// TIA Portal V18 program export: 1 tag tables, 1 data types, 4 data blocks, 17 code blocks (in call order from the OBs), 10 instance data blocks

VAR_GLOBAL   // PLC tag table "默认变量表"
   System_Byte AT %MB1 : Byte;
   FirstScan AT %M1.0 : Bool;
   DiagStatusUpdate AT %M1.1 : Bool;
   AlwaysTRUE AT %M1.2 : Bool;
   AlwaysFALSE AT %M1.3 : Bool;
   Clock_Byte AT %MB0 : Byte;
   Clock_10Hz AT %M0.0 : Bool;
   Clock_5Hz AT %M0.1 : Bool;
   "Clock_2.5Hz" AT %M0.2 : Bool;
   Clock_2Hz AT %M0.3 : Bool;
   "Clock_1.25Hz" AT %M0.4 : Bool;
   Clock_1Hz AT %M0.5 : Bool;
   "Clock_0.625Hz" AT %M0.6 : Bool;
   "Clock_0.5Hz" AT %M0.7 : Bool;
END_VAR

TYPE "FIODia"
// stored: IsFailsafeCompliant true
   STRUCT
      ModulePassOut : Bool;   // 模块钝化
      ModuleACK_REQ : Bool;   // 模块需确认重新集成
      Channel0PassOut : Bool;   // 通道0钝化
      Channel1PassOut : Bool;   // 通道1钝化
      Channel2PassOut : Bool;   // 通道2钝化
      Channel3PassOut : Bool;   // 通道3钝化
      Channel4PassOut : Bool;   // 通道4钝化
      Channel5PassOut : Bool;   // 通道5钝化
      Channel6PassOut : Bool;   // 通道6钝化
      Channel7PassOut : Bool;   // 通道7钝化
   END_STRUCT;
END_TYPE

DATA_BLOCK "TCSData"   // DB4
{ S7_Optimized_Access := 'TRUE' }
VERSION : 0.1
// stored: AutoNumber true, DBAccessibleFromOPCUA true, IsOnlyStoredInLoadMemory false, IsRetainMemResEnabled false, IsWriteProtectedInAS false, MemoryReserve 100
   VAR
      Data : Array[0..1] of Word;
      Connect : TCON_IP_v4;
   END_VAR
BEGIN
   Connect.InterfaceId := 64;
   Connect.ID := 16#1;
   Connect.LocalPort := 502;
END_DATA_BLOCK

DATA_BLOCK "数据块_1"   // DB2
{ S7_Optimized_Access := 'TRUE' }
VERSION : 0.1
// stored: AutoNumber true, DBAccessibleFromOPCUA true, IsOnlyStoredInLoadMemory false, IsRetainMemResEnabled false, IsWriteProtectedInAS false, MemoryReserve 100
   VAR
      Room1_Interlock : Bool;
      Room2_Interlock : Bool;
      ACC_Interlock : Bool;
      VerticalBeam_Interlock : Bool;
      Interlock : Bool;
   END_VAR
BEGIN
END_DATA_BLOCK

DATA_BLOCK "数据块_2"   // DB3
{ S7_Optimized_Access := 'TRUE' }
VERSION : 0.1
// stored: AutoNumber true, DBAccessibleFromOPCUA true, IsOnlyStoredInLoadMemory false, IsRetainMemResEnabled false, IsWriteProtectedInAS false, MemoryReserve 100
   VAR
      "F-DI_A21_1" : "FIODia";   // 安全输入模块A21.1
      "F-DI_A21_2" { S7_SetPoint := 'True'} : "FIODia";   // 安全输入模块A21.2
      "F-DI_A21_3" { S7_SetPoint := 'True'} : "FIODia";   // 安全输入模块A21.3
      "F-DI_A21_4" { S7_SetPoint := 'True'} : "FIODia";   // 安全输入模块A21.4
      "F-DI_A21_5" { S7_SetPoint := 'True'} : "FIODia";   // 安全输入模块A21.5
      "F-DI_A21_6" { S7_SetPoint := 'True'} : "FIODia";   // 安全输入模块A21.6
      "F-DI_A21_7" { S7_SetPoint := 'True'} : "FIODia";   // 安全输入模块A21.7
      "F-DI_A21_8" { S7_SetPoint := 'True'} : "FIODia";   // 安全输入模块A21.8
      "F-DI_A21_9" { S7_SetPoint := 'True'} : "FIODia";   // 安全输入模块A21.9
      "F-DI_A21_10" { S7_SetPoint := 'True'} : "FIODia";   // 安全输入模块A21.10
      "F-DI_A21_11" { S7_SetPoint := 'True'} : "FIODia";   // 安全输入模块A21.11
      "F-DI_A21_12" { S7_SetPoint := 'True'} : "FIODia";   // 安全输入模块A21.12
      "F-DQ_A21_1" { S7_SetPoint := 'True'} : "FIODia";   // 安全输出模块A22.1
      "F-DQ_A21_2" { S7_SetPoint := 'True'} : "FIODia";   // 安全输出模块A22.2
   END_VAR
BEGIN
END_DATA_BLOCK

DATA_BLOCK "EPICSData"   // DB8
{ S7_Optimized_Access := 'FALSE'; DB_Accessible_From_OPC_UA := 'FALSE' }
VERSION : 0.1
// stored: AutoNumber true, DBAccessibleFromOPCUA false, IsOnlyStoredInLoadMemory false, IsWriteProtectedInAS false
   VAR
      Reset : Bool;
   END_VAR
BEGIN
END_DATA_BLOCK

ORGANIZATION_BLOCK "Main"   // OB1, LAD, ProgramCycle
TITLE = "Main Program Sweep (Cycle)"
{ S7_Optimized_Access := 'TRUE' }
VERSION : 0.1
// stored: AutoNumber true, IsIECCheckEnabled false, SetENOAutomatically false
   VAR_INPUT
      Initial_Call : Bool;   // Initial call of this OB
      Remanence : Bool;   // =True, if remanent data are available
   END_VAR
BEGIN

REGION Network 1: 11
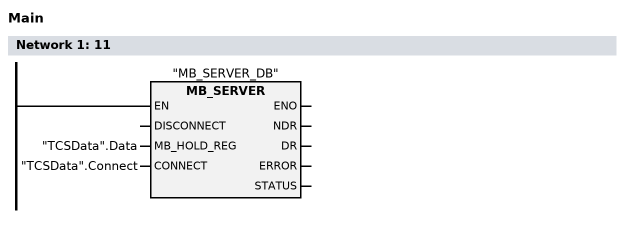
   RUNG wire#powerrail
      "MB_SERVER_DB".MB_SERVER(DISCONNECT :=, MB_HOLD_REG := "TCSData".Data, CONNECT := "TCSData".Connect, NDR =>, DR =>, ERROR =>, STATUS =>)
   END_RUNG
   // the same network as SCL:
   "MB_SERVER_DB"(MB_HOLD_REG := "TCSData".Data, CONNECT := "TCSData".Connect);   // MB_SERVER
END_REGION
END_ORGANIZATION_BLOCK

ORGANIZATION_BLOCK "Time error interrupt"   // OB80, LAD, TimeErrorInterrupt
{ S7_Optimized_Access := 'TRUE' }
VERSION : 0.1
// stored: IsIECCheckEnabled false, SetENOAutomatically false
   VAR_INPUT
      Fault_ID : Byte;   // Fault identifier
      Csg_OBnr : OB_ANY;   // Number of OB causing the error
      Csg_Prio : UInt;   // Priority of OB causing the error
   END_VAR
BEGIN
END_ORGANIZATION_BLOCK

FUNCTION_BLOCK "AccessControl"   // FB7, LAD
{ S7_Optimized_Access := 'TRUE' }
VERSION : 0.1
// stored: AutoNumber true, IsIECCheckEnabled false, IsRetainMemResEnabled false, MemoryReserve 100, SetENOAutomatically false, UDAEnableTagReadback false
   VAR_INPUT
      SearchStatus : Int;   // 0:未搜索;1:搜索中;2:搜索完成;
      RunArea : Bool;
      ACC_Ready : Bool;
      ACC_Run : Bool;
      ACC_StopBeam : Bool;
      Key : Bool;
      keyControl : Bool;
      Interlock : Bool;
      DoseAttenuation_Time : Time := T#1m;
      StartAlarm_Time : Time := T#2m;
   END_VAR
   VAR_OUTPUT
      StartAlarm : Bool;
      NoEntry : Bool;
      RestrictedEntry : Bool;
      ControlEntry : Bool;
   END_VAR
   VAR_IN_OUT
      AreaReady : Bool;
      BeamAllowed : Bool;
   END_VAR
   VAR
      State : Int;   // 0:禁止进入;1:限制进入;2:控制进入
      DoseAttenuation_Timer { S7_SetPoint := 'True'} : TON_TIME;
      StartAlarm_Timer { S7_SetPoint := 'True'} : TON_TIME;
   END_VAR
   VAR_TEMP   // added for the SCL form of the ladder/FBD networks
      _w1 : Bool;
   END_VAR
BEGIN

REGION Network 1
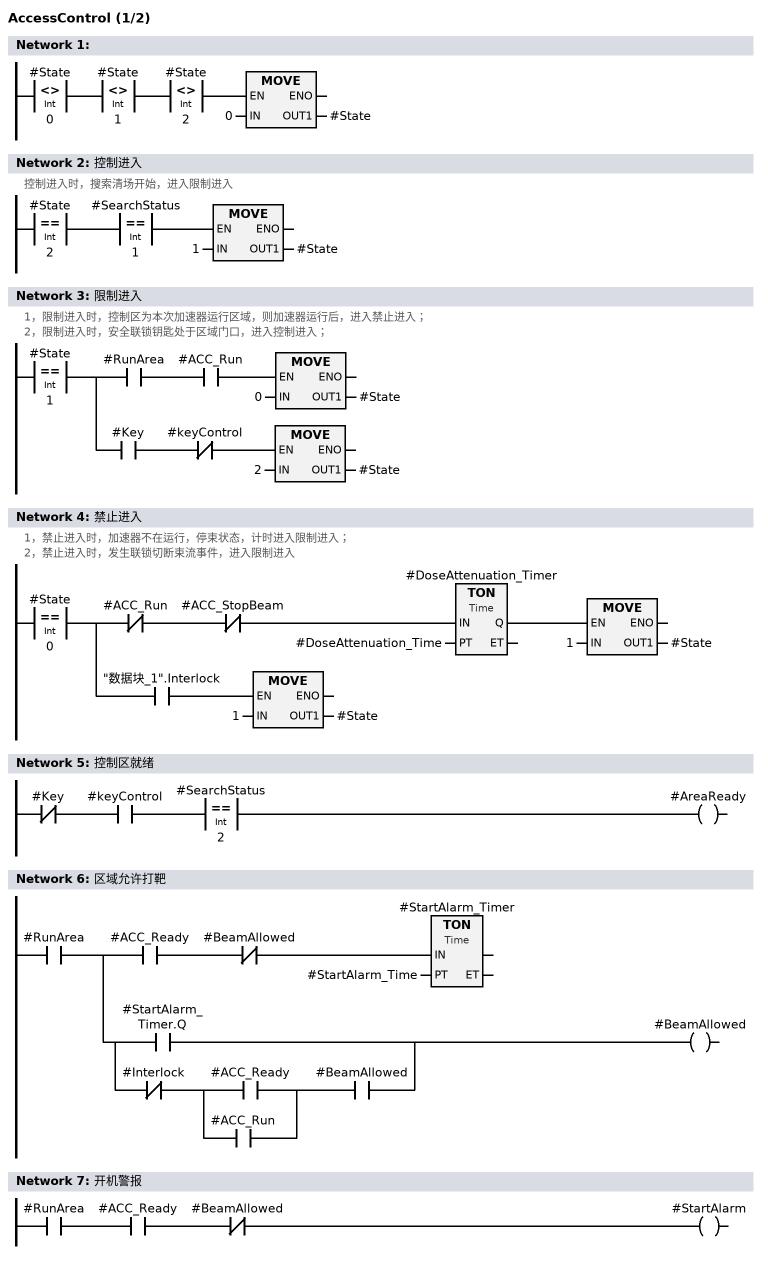
   RUNG wire#powerrail
      { S7_Templates := "SrcType := Int" } NE_Contact(in1 := #State, in2 := 0)
      { S7_Templates := "SrcType := Int" } NE_Contact(in1 := #State, in2 := 1)
      { S7_Templates := "SrcType := Int" } NE_Contact(in1 := #State, in2 := 2)
      Move(in := 0, out1 => #State)
   END_RUNG
   // the same network as SCL:
   IF (#State <> 0) AND (#State <> 1) AND (#State <> 2) THEN #State := 0; END_IF;
END_REGION

REGION Network 2: 控制进入
   // 控制进入时，搜索清场开始，进入限制进入
   RUNG wire#powerrail
      { S7_Templates := "SrcType := Int" } EQ_Contact(in1 := #State, in2 := 2)
      { S7_Templates := "SrcType := Int" } EQ_Contact(in1 := #SearchStatus, in2 := 1)
      Move(in := 1, out1 => #State)
   END_RUNG
   // the same network as SCL:
   IF (#State = 2) AND (#SearchStatus = 1) THEN #State := 1; END_IF;
END_REGION

REGION Network 3: 限制进入
   // 1，限制进入时，控制区为本次加速器运行区域，则加速器运行后，进入禁止进入；
   // 2，限制进入时，安全联锁钥匙处于区域门口，进入控制进入；
   RUNG wire#powerrail
      { S7_Templates := "SrcType := Int" } EQ_Contact(in1 := #State, in2 := 1)
      wire#w1
      Contact( #RunArea )
      Contact( #ACC_Run )
      Move(in := 0, out1 => #State)
   END_RUNG
   RUNG wire#w1
      Contact( #Key )
      I_Contact( #keyControl )
      Move(in := 2, out1 => #State)
   END_RUNG
   // the same network as SCL:
   #_w1 := #State = 1;
   IF #_w1 AND #RunArea AND #ACC_Run THEN #State := 0; END_IF;
   IF #_w1 AND #Key AND NOT #keyControl THEN #State := 2; END_IF;
END_REGION

REGION Network 4: 禁止进入
   // 1，禁止进入时，加速器不在运行，停束状态，计时进入限制进入；
   // 2，禁止进入时，发生联锁切断束流事件，进入限制进入
   RUNG wire#powerrail
      { S7_Templates := "SrcType := Int" } EQ_Contact(in1 := #State, in2 := 0)
      wire#w1
      I_Contact( #ACC_Run )
      I_Contact( #ACC_StopBeam )
      { S7_Templates := "time_type := Time" } #DoseAttenuation_Timer.TON(pt := #DoseAttenuation_Time, et =>)
      Move(in := 1, out1 => #State)
   END_RUNG
   RUNG wire#w1
      Contact( "数据块_1".Interlock )
      Move(in := 1, out1 => #State)
   END_RUNG
   // the same network as SCL:
   #_w1 := #State = 0;
   #DoseAttenuation_Timer(IN := #_w1 AND NOT #ACC_Run AND NOT #ACC_StopBeam, PT := #DoseAttenuation_Time);   // TON
   IF #DoseAttenuation_Timer.Q THEN #State := 1; END_IF;
   IF #_w1 AND "数据块_1".Interlock THEN #State := 1; END_IF;
END_REGION

REGION Network 5: 控制区就绪
   RUNG wire#powerrail
      I_Contact( #Key )
      Contact( #keyControl )
      { S7_Templates := "SrcType := Int" } EQ_Contact(in1 := #SearchStatus, in2 := 2)
      Coil( #AreaReady )
   END_RUNG
   // the same network as SCL:
   #AreaReady := NOT #Key AND #keyControl AND (#SearchStatus = 2);
END_REGION

REGION Network 6: 区域允许打靶
   RUNG wire#powerrail
      Contact( #RunArea )
      wire#w1
      Contact( #ACC_Ready )
      I_Contact( #BeamAllowed )
      { S7_Templates := "time_type := Time" } #StartAlarm_Timer.TON(pt := #StartAlarm_Time, et =>)
   END_RUNG
   RUNG wire#w1
      Contact( #StartAlarm_Timer.Q )
      wire#w2
      Coil( #BeamAllowed )
   END_RUNG
   RUNG wire#w1
      I_Contact( #Interlock )
      wire#w3
      Contact( #ACC_Ready )
      wire#w4
      Contact( #BeamAllowed )
   END_RUNG wire#w2
   RUNG wire#w3
      Contact( #ACC_Run )
   END_RUNG wire#w4
   // the same network as SCL:
   #StartAlarm_Timer(IN := #RunArea AND #ACC_Ready AND NOT #BeamAllowed, PT := #StartAlarm_Time);   // TON
   #BeamAllowed := #RunArea AND (#StartAlarm_Timer.Q OR (NOT #Interlock AND (#ACC_Ready OR #ACC_Run) AND #BeamAllowed));
END_REGION

REGION Network 7: 开机警报
   RUNG wire#powerrail
      Contact( #RunArea )
      Contact( #ACC_Ready )
      I_Contact( #BeamAllowed )
      Coil( #StartAlarm )
   END_RUNG
   // the same network as SCL:
   #StartAlarm := #RunArea AND #ACC_Ready AND NOT #BeamAllowed;
END_REGION

REGION Network 8
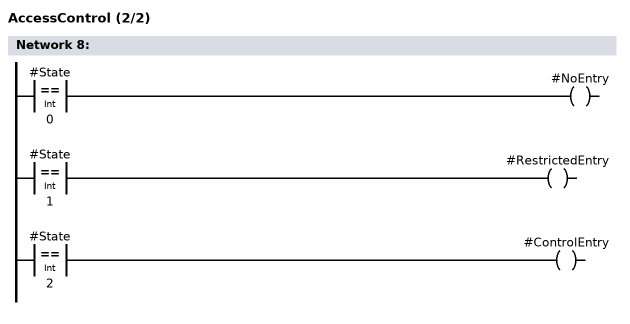
   RUNG wire#powerrail
      { S7_Templates := "SrcType := Int" } EQ_Contact(in1 := #State, in2 := 0)
      Coil( #NoEntry )
   END_RUNG
   RUNG wire#powerrail
      { S7_Templates := "SrcType := Int" } EQ_Contact(in1 := #State, in2 := 1)
      Coil( #RestrictedEntry )
   END_RUNG
   RUNG wire#powerrail
      { S7_Templates := "SrcType := Int" } EQ_Contact(in1 := #State, in2 := 2)
      Coil( #ControlEntry )
   END_RUNG
   // the same network as SCL:
   #NoEntry := #State = 0;
   #RestrictedEntry := #State = 1;
   #ControlEntry := #State = 2;
END_REGION
END_FUNCTION_BLOCK

FUNCTION_BLOCK "SearchArea"   // FB6, LAD
{ S7_Optimized_Access := 'TRUE' }
VERSION : 0.1
// stored: AutoNumber true, IsIECCheckEnabled false, IsRetainMemResEnabled false, MemoryReserve 100, SetENOAutomatically false, UDAEnableTagReadback false
   VAR_INPUT
      SB1 : Bool;
      SB2 : Bool;
      Door : Bool;
      "E-Stop" : Bool;
      SearchArea_Time : Time := T#5m;
      Reset : Bool;
   END_VAR
   VAR
      SearchArea_Timer { S7_SetPoint := 'True'} : TON_TIME;
      SearchArea_Status : Int;   // 0:未搜索;1:搜索中;2:搜索完成;
      "Step" { S7_SetPoint := 'True'} : Int;
      Error { ExternalAccessible := 'False'; ExternalVisible := 'False'; ExternalWritable := 'False'} : Struct
         All { ExternalAccessible := 'False'; ExternalVisible := 'False'; ExternalWritable := 'False'} : Bool;   // 搜索总故障
         StartFail { ExternalAccessible := 'False'; ExternalVisible := 'False'; ExternalWritable := 'False'} : Bool;   // 搜索启动失败，请确认未按下搜索按钮2或未关闭门
         WrongSequence1 { ExternalAccessible := 'False'; ExternalVisible := 'False'; ExternalWritable := 'False'} : Bool;   // 搜索顺序错误，此时应按下搜索按钮2，请勿按搜索按钮1或关闭门
         WrongSequence2 { ExternalAccessible := 'False'; ExternalVisible := 'False'; ExternalWritable := 'False'} : Bool;   // 搜索顺序错误，此时应关闭门，请勿按搜索按钮1或搜索按钮2
         Timeout { ExternalAccessible := 'False'; ExternalVisible := 'False'; ExternalWritable := 'False'} : Bool;   // 搜索超时
      END_STRUCT;
   END_VAR
   VAR_TEMP   // added for the SCL form of the ladder/FBD networks
      _w1 : Bool;
   END_VAR
BEGIN

REGION Network 1: 搜索破坏
   // 搜索完成后，当搜索按钮按下，门被打开，急停按钮按下，搜索状态设置为未搜索
   // 需与客户确认破坏条件是否包含搜索按钮和急停？
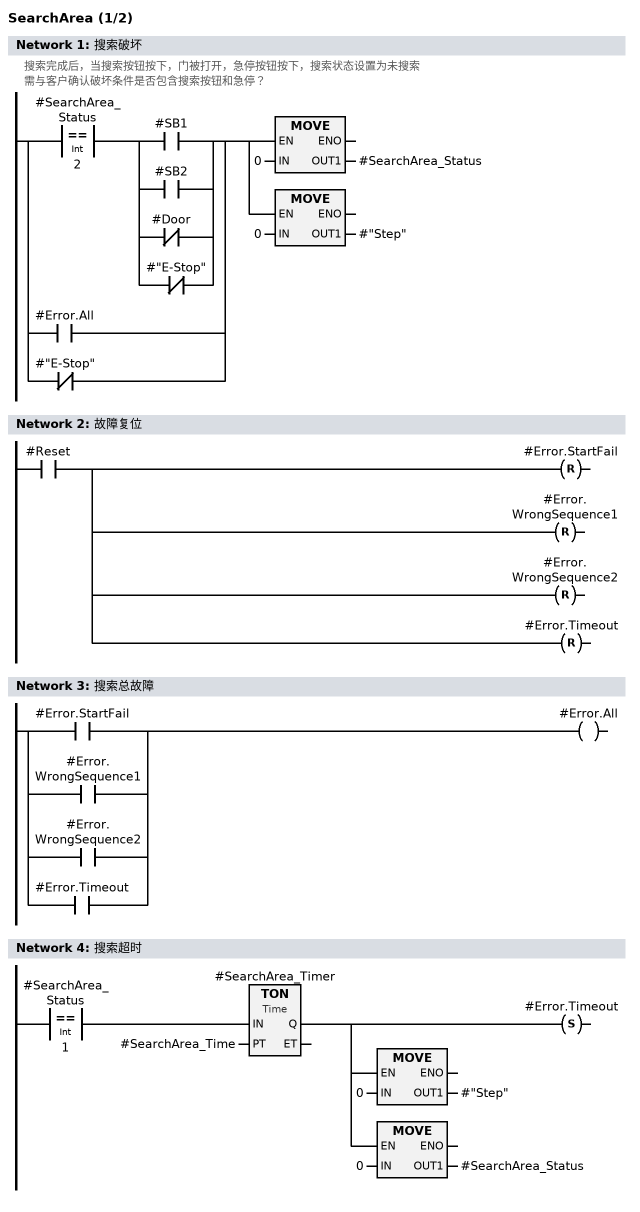
   RUNG wire#powerrail
      { S7_Templates := "SrcType := Int" } EQ_Contact(in1 := #SearchArea_Status, in2 := 2)
      wire#w1
      Contact( #SB1 )
      wire#w2
      Move(in := 0, out1 => #SearchArea_Status)
   END_RUNG
   RUNG wire#w1
      Contact( #SB2 )
   END_RUNG wire#w2
   RUNG wire#w1
      I_Contact( #Door )
   END_RUNG wire#w2
   RUNG wire#w1
      I_Contact( #"E-Stop" )
   END_RUNG wire#w2
   RUNG wire#powerrail
      Contact( #Error.All )
   END_RUNG wire#w2
   RUNG wire#powerrail
      I_Contact( #"E-Stop" )
   END_RUNG wire#w2
   RUNG wire#w2
      Move(in := 0, out1 => #"Step")
   END_RUNG
   // the same network as SCL:
   #_w1 := ((#SearchArea_Status = 2) AND (#SB1 OR #SB2 OR NOT #Door OR NOT #"E-Stop")) OR #Error.All OR NOT #"E-Stop";
   IF #_w1 THEN
       #SearchArea_Status := 0;
       #"Step" := 0;
   END_IF;
END_REGION

REGION Network 2: 故障复位
   RUNG wire#powerrail
      Contact( #Reset )
      wire#w1
      R_Coil( #Error.StartFail )
   END_RUNG
   RUNG wire#w1
      R_Coil( #Error.WrongSequence1 )
   END_RUNG
   RUNG wire#w1
      R_Coil( #Error.WrongSequence2 )
   END_RUNG
   RUNG wire#w1
      R_Coil( #Error.Timeout )
   END_RUNG
   // the same network as SCL:
   IF #Reset THEN
       #Error.StartFail := FALSE;
       #Error.WrongSequence1 := FALSE;
       #Error.WrongSequence2 := FALSE;
       #Error.Timeout := FALSE;
   END_IF;
END_REGION

REGION Network 3: 搜索总故障
   RUNG wire#powerrail
      Contact( #Error.StartFail )
      wire#w1
      Coil( #Error.All )
   END_RUNG
   RUNG wire#powerrail
      Contact( #Error.WrongSequence1 )
   END_RUNG wire#w1
   RUNG wire#powerrail
      Contact( #Error.WrongSequence2 )
   END_RUNG wire#w1
   RUNG wire#powerrail
      Contact( #Error.Timeout )
   END_RUNG wire#w1
   // the same network as SCL:
   #Error.All := #Error.StartFail OR #Error.WrongSequence1 OR #Error.WrongSequence2 OR #Error.Timeout;
END_REGION

REGION Network 4: 搜索超时
   RUNG wire#powerrail
      { S7_Templates := "SrcType := Int" } EQ_Contact(in1 := #SearchArea_Status, in2 := 1)
      { S7_Templates := "time_type := Time" } #SearchArea_Timer.TON(pt := #SearchArea_Time, et =>)
      wire#w1
      S_Coil( #Error.Timeout )
   END_RUNG
   RUNG wire#w1
      Move(in := 0, out1 => #"Step")
   END_RUNG
   RUNG wire#w1
      Move(in := 0, out1 => #SearchArea_Status)
   END_RUNG
   // the same network as SCL:
   #SearchArea_Timer(IN := #SearchArea_Status = 1, PT := #SearchArea_Time);   // TON
   IF #SearchArea_Timer.Q THEN
       #Error.Timeout := TRUE;
       #"Step" := 0;
       #SearchArea_Status := 0;
   END_IF;
END_REGION

REGION Network 5: 按下SB1，开始搜索
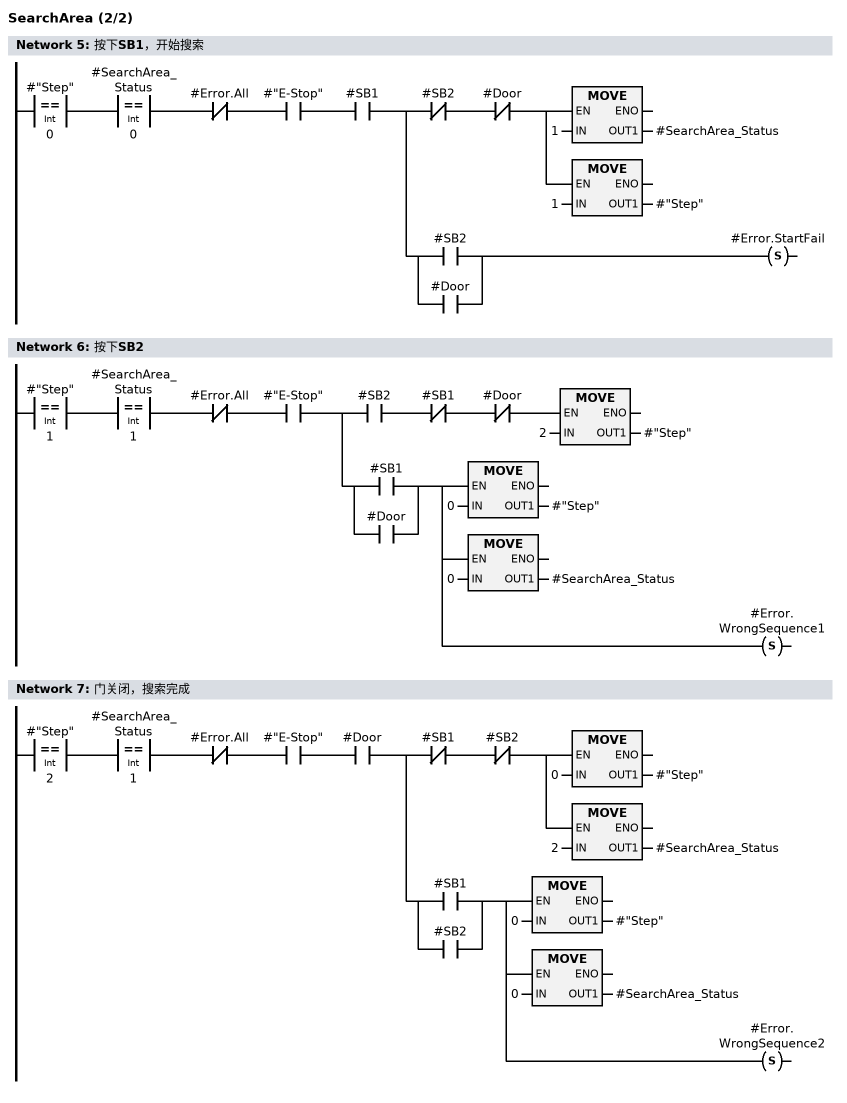
   RUNG wire#powerrail
      { S7_Templates := "SrcType := Int" } EQ_Contact(in1 := #"Step", in2 := 0)
      { S7_Templates := "SrcType := Int" } EQ_Contact(in1 := #SearchArea_Status, in2 := 0)
      I_Contact( #Error.All )
      Contact( #"E-Stop" )
      Contact( #SB1 )
      wire#w1
      I_Contact( #SB2 )
      I_Contact( #Door )
      wire#w2
      Move(in := 1, out1 => #SearchArea_Status)
   END_RUNG
   RUNG wire#w2
      Move(in := 1, out1 => #"Step")
   END_RUNG
   RUNG wire#w1
      Contact( #SB2 )
      wire#w3
      S_Coil( #Error.StartFail )
   END_RUNG
   RUNG wire#w1
      Contact( #Door )
   END_RUNG wire#w3
   // the same network as SCL:
   #_w1 := (#"Step" = 0) AND (#SearchArea_Status = 0) AND NOT #Error.All AND #"E-Stop" AND #SB1;
   IF #_w1 AND NOT #SB2 AND NOT #Door THEN
       #SearchArea_Status := 1;
       #"Step" := 1;
   END_IF;
   IF #_w1 AND (#SB2 OR #Door) THEN #Error.StartFail := TRUE; END_IF;
END_REGION

REGION Network 6: 按下SB2
   RUNG wire#powerrail
      { S7_Templates := "SrcType := Int" } EQ_Contact(in1 := #"Step", in2 := 1)
      { S7_Templates := "SrcType := Int" } EQ_Contact(in1 := #SearchArea_Status, in2 := 1)
      I_Contact( #Error.All )
      Contact( #"E-Stop" )
      wire#w1
      Contact( #SB2 )
      I_Contact( #SB1 )
      I_Contact( #Door )
      Move(in := 2, out1 => #"Step")
   END_RUNG
   RUNG wire#w1
      Contact( #SB1 )
      wire#w2
      Move(in := 0, out1 => #"Step")
   END_RUNG
   RUNG wire#w1
      Contact( #Door )
   END_RUNG wire#w2
   RUNG wire#w2
      Move(in := 0, out1 => #SearchArea_Status)
   END_RUNG
   RUNG wire#w2
      S_Coil( #Error.WrongSequence1 )
   END_RUNG
   // the same network as SCL:
   #_w1 := (#"Step" = 1) AND (#SearchArea_Status = 1) AND NOT #Error.All AND #"E-Stop";
   IF #_w1 AND #SB2 AND NOT #SB1 AND NOT #Door THEN #"Step" := 2; END_IF;
   IF #_w1 AND (#SB1 OR #Door) THEN
       #"Step" := 0;
       #SearchArea_Status := 0;
       #Error.WrongSequence1 := TRUE;
   END_IF;
END_REGION

REGION Network 7: 门关闭，搜索完成
   RUNG wire#powerrail
      { S7_Templates := "SrcType := Int" } EQ_Contact(in1 := #"Step", in2 := 2)
      { S7_Templates := "SrcType := Int" } EQ_Contact(in1 := #SearchArea_Status, in2 := 1)
      I_Contact( #Error.All )
      Contact( #"E-Stop" )
      Contact( #Door )
      wire#w1
      I_Contact( #SB1 )
      I_Contact( #SB2 )
      wire#w2
      Move(in := 0, out1 => #"Step")
   END_RUNG
   RUNG wire#w2
      Move(in := 2, out1 => #SearchArea_Status)
   END_RUNG
   RUNG wire#w1
      Contact( #SB1 )
      wire#w3
      Move(in := 0, out1 => #"Step")
   END_RUNG
   RUNG wire#w1
      Contact( #SB2 )
   END_RUNG wire#w3
   RUNG wire#w3
      Move(in := 0, out1 => #SearchArea_Status)
   END_RUNG
   RUNG wire#w3
      S_Coil( #Error.WrongSequence2 )
   END_RUNG
   // the same network as SCL:
   #_w1 := (#"Step" = 2) AND (#SearchArea_Status = 1) AND NOT #Error.All AND #"E-Stop" AND #Door;
   IF #_w1 AND NOT #SB1 AND NOT #SB2 THEN
       #"Step" := 0;
       #SearchArea_Status := 2;
   END_IF;
   IF #_w1 AND (#SB1 OR #SB2) THEN
       #"Step" := 0;
       #SearchArea_Status := 0;
       #Error.WrongSequence2 := TRUE;
   END_IF;
END_REGION
END_FUNCTION_BLOCK

FUNCTION_BLOCK "SearchArea_2doors"   // FB8, LAD
{ S7_Optimized_Access := 'TRUE' }
VERSION : 0.1
// stored: AutoNumber true, IsIECCheckEnabled false, IsRetainMemResEnabled false, MemoryReserve 100, SetENOAutomatically false, UDAEnableTagReadback false
   VAR_INPUT
      SB1 : Bool;
      SB2 : Bool;
      Door1 : Bool;
      Door2 : Bool;
      "E-Stop" : Bool;
      SearchArea_Time : Time := T#5m;
      Reset : Bool;
   END_VAR
   VAR
      SearchArea_Timer { S7_SetPoint := 'True'} : TON_TIME;
      SearchArea_Status : Int;   // 0:未搜索;1:搜索中;2:搜索完成;
      "Step" { S7_SetPoint := 'True'} : Int;
      Error { ExternalAccessible := 'False'; ExternalVisible := 'False'; ExternalWritable := 'False'} : Struct
         All { ExternalAccessible := 'False'; ExternalVisible := 'False'; ExternalWritable := 'False'} : Bool;   // 搜索总故障
         StartFail { ExternalAccessible := 'False'; ExternalVisible := 'False'; ExternalWritable := 'False'} : Bool;   // 搜索启动失败，请确认未按下搜索按钮2或未关闭门1或门2
         WrongSequence1 { ExternalAccessible := 'False'; ExternalVisible := 'False'; ExternalWritable := 'False'} : Bool;   // 搜索顺序错误，此时应按下搜索按钮2，请勿按搜索按钮1或关闭门1或门2
         WrongSequence2 { ExternalAccessible := 'False'; ExternalVisible := 'False'; ExternalWritable := 'False'} : Bool;   // 搜索顺序错误，此时应关闭门1，请勿按搜索按钮1或搜索按钮2或门2
         WrongSequence3 { ExternalAccessible := 'False'; ExternalVisible := 'False'; ExternalWritable := 'False'} : Bool;   // 搜索顺序错误，此时应关闭门2，请勿按搜索按钮1或搜索按钮2或打开门1
         Timeout { ExternalAccessible := 'False'; ExternalVisible := 'False'; ExternalWritable := 'False'} : Bool;   // 搜索超时
      END_STRUCT;
   END_VAR
   VAR_TEMP   // added for the SCL form of the ladder/FBD networks
      _w1 : Bool;
   END_VAR
BEGIN

REGION Network 1: 搜索破坏
   // 搜索完成后，当搜索按钮按下，门被打开，急停按钮按下，搜索状态设置为未搜索
   // 需与客户确认破坏条件是否包含搜索按钮和急停？
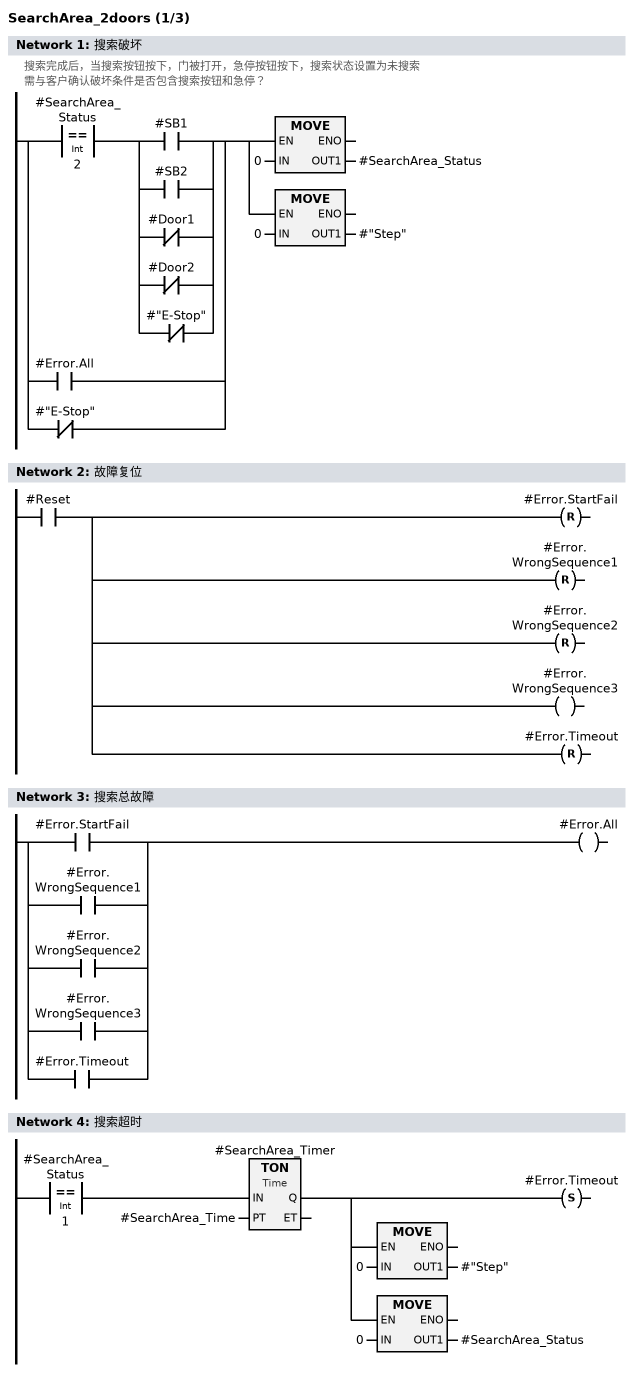
   RUNG wire#powerrail
      { S7_Templates := "SrcType := Int" } EQ_Contact(in1 := #SearchArea_Status, in2 := 2)
      wire#w1
      Contact( #SB1 )
      wire#w2
      Move(in := 0, out1 => #SearchArea_Status)
   END_RUNG
   RUNG wire#w1
      Contact( #SB2 )
   END_RUNG wire#w2
   RUNG wire#w1
      I_Contact( #Door1 )
   END_RUNG wire#w2
   RUNG wire#w1
      I_Contact( #Door2 )
   END_RUNG wire#w2
   RUNG wire#w1
      I_Contact( #"E-Stop" )
   END_RUNG wire#w2
   RUNG wire#powerrail
      Contact( #Error.All )
   END_RUNG wire#w2
   RUNG wire#powerrail
      I_Contact( #"E-Stop" )
   END_RUNG wire#w2
   RUNG wire#w2
      Move(in := 0, out1 => #"Step")
   END_RUNG
   // the same network as SCL:
   #_w1 := ((#SearchArea_Status = 2) AND (#SB1 OR #SB2 OR NOT #Door1 OR NOT #Door2 OR NOT #"E-Stop")) OR #Error.All OR NOT #"E-Stop";
   IF #_w1 THEN
       #SearchArea_Status := 0;
       #"Step" := 0;
   END_IF;
END_REGION

REGION Network 2: 故障复位
   RUNG wire#powerrail
      Contact( #Reset )
      wire#w1
      R_Coil( #Error.StartFail )
   END_RUNG
   RUNG wire#w1
      R_Coil( #Error.WrongSequence1 )
   END_RUNG
   RUNG wire#w1
      R_Coil( #Error.WrongSequence2 )
   END_RUNG
   RUNG wire#w1
      Coil( #Error.WrongSequence3 )
   END_RUNG
   RUNG wire#w1
      R_Coil( #Error.Timeout )
   END_RUNG
   // the same network as SCL:
   IF #Reset THEN
       #Error.StartFail := FALSE;
       #Error.WrongSequence1 := FALSE;
       #Error.WrongSequence2 := FALSE;
   END_IF;
   #Error.WrongSequence3 := #Reset;
   IF #Reset THEN #Error.Timeout := FALSE; END_IF;
END_REGION

REGION Network 3: 搜索总故障
   RUNG wire#powerrail
      Contact( #Error.StartFail )
      wire#w1
      Coil( #Error.All )
   END_RUNG
   RUNG wire#powerrail
      Contact( #Error.WrongSequence1 )
   END_RUNG wire#w1
   RUNG wire#powerrail
      Contact( #Error.WrongSequence2 )
   END_RUNG wire#w1
   RUNG wire#powerrail
      Contact( #Error.WrongSequence3 )
   END_RUNG wire#w1
   RUNG wire#powerrail
      Contact( #Error.Timeout )
   END_RUNG wire#w1
   // the same network as SCL:
   #Error.All := #Error.StartFail OR #Error.WrongSequence1 OR #Error.WrongSequence2 OR #Error.WrongSequence3 OR #Error.Timeout;
END_REGION

REGION Network 4: 搜索超时
   RUNG wire#powerrail
      { S7_Templates := "SrcType := Int" } EQ_Contact(in1 := #SearchArea_Status, in2 := 1)
      { S7_Templates := "time_type := Time" } #SearchArea_Timer.TON(pt := #SearchArea_Time, et =>)
      wire#w1
      S_Coil( #Error.Timeout )
   END_RUNG
   RUNG wire#w1
      Move(in := 0, out1 => #"Step")
   END_RUNG
   RUNG wire#w1
      Move(in := 0, out1 => #SearchArea_Status)
   END_RUNG
   // the same network as SCL:
   #SearchArea_Timer(IN := #SearchArea_Status = 1, PT := #SearchArea_Time);   // TON
   IF #SearchArea_Timer.Q THEN
       #Error.Timeout := TRUE;
       #"Step" := 0;
       #SearchArea_Status := 0;
   END_IF;
END_REGION

REGION Network 5: 按下SB1，开始搜索
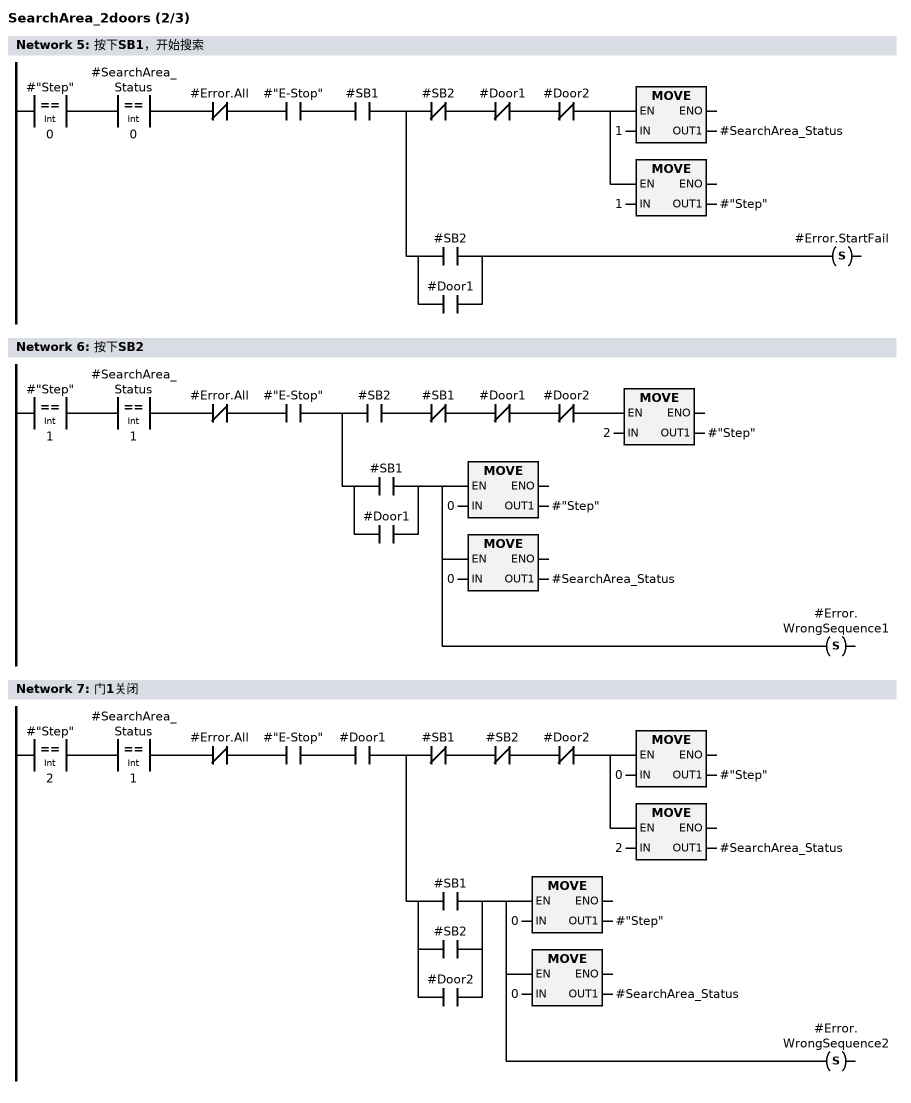
   RUNG wire#powerrail
      { S7_Templates := "SrcType := Int" } EQ_Contact(in1 := #"Step", in2 := 0)
      { S7_Templates := "SrcType := Int" } EQ_Contact(in1 := #SearchArea_Status, in2 := 0)
      I_Contact( #Error.All )
      Contact( #"E-Stop" )
      Contact( #SB1 )
      wire#w1
      I_Contact( #SB2 )
      I_Contact( #Door1 )
      I_Contact( #Door2 )
      wire#w2
      Move(in := 1, out1 => #SearchArea_Status)
   END_RUNG
   RUNG wire#w2
      Move(in := 1, out1 => #"Step")
   END_RUNG
   RUNG wire#w1
      Contact( #SB2 )
      wire#w3
      S_Coil( #Error.StartFail )
   END_RUNG
   RUNG wire#w1
      Contact( #Door1 )
   END_RUNG wire#w3
   // the same network as SCL:
   #_w1 := (#"Step" = 0) AND (#SearchArea_Status = 0) AND NOT #Error.All AND #"E-Stop" AND #SB1;
   IF #_w1 AND NOT #SB2 AND NOT #Door1 AND NOT #Door2 THEN
       #SearchArea_Status := 1;
       #"Step" := 1;
   END_IF;
   IF #_w1 AND (#SB2 OR #Door1) THEN #Error.StartFail := TRUE; END_IF;
END_REGION

REGION Network 6: 按下SB2
   RUNG wire#powerrail
      { S7_Templates := "SrcType := Int" } EQ_Contact(in1 := #"Step", in2 := 1)
      { S7_Templates := "SrcType := Int" } EQ_Contact(in1 := #SearchArea_Status, in2 := 1)
      I_Contact( #Error.All )
      Contact( #"E-Stop" )
      wire#w1
      Contact( #SB2 )
      I_Contact( #SB1 )
      I_Contact( #Door1 )
      I_Contact( #Door2 )
      Move(in := 2, out1 => #"Step")
   END_RUNG
   RUNG wire#w1
      Contact( #SB1 )
      wire#w2
      Move(in := 0, out1 => #"Step")
   END_RUNG
   RUNG wire#w1
      Contact( #Door1 )
   END_RUNG wire#w2
   RUNG wire#w2
      Move(in := 0, out1 => #SearchArea_Status)
   END_RUNG
   RUNG wire#w2
      S_Coil( #Error.WrongSequence1 )
   END_RUNG
   // the same network as SCL:
   #_w1 := (#"Step" = 1) AND (#SearchArea_Status = 1) AND NOT #Error.All AND #"E-Stop";
   IF #_w1 AND #SB2 AND NOT #SB1 AND NOT #Door1 AND NOT #Door2 THEN #"Step" := 2; END_IF;
   IF #_w1 AND (#SB1 OR #Door1) THEN
       #"Step" := 0;
       #SearchArea_Status := 0;
       #Error.WrongSequence1 := TRUE;
   END_IF;
END_REGION

REGION Network 7: 门1关闭
   RUNG wire#powerrail
      { S7_Templates := "SrcType := Int" } EQ_Contact(in1 := #"Step", in2 := 2)
      { S7_Templates := "SrcType := Int" } EQ_Contact(in1 := #SearchArea_Status, in2 := 1)
      I_Contact( #Error.All )
      Contact( #"E-Stop" )
      Contact( #Door1 )
      wire#w1
      I_Contact( #SB1 )
      I_Contact( #SB2 )
      I_Contact( #Door2 )
      wire#w2
      Move(in := 0, out1 => #"Step")
   END_RUNG
   RUNG wire#w2
      Move(in := 2, out1 => #SearchArea_Status)
   END_RUNG
   RUNG wire#w1
      Contact( #SB1 )
      wire#w3
      Move(in := 0, out1 => #"Step")
   END_RUNG
   RUNG wire#w1
      Contact( #SB2 )
   END_RUNG wire#w3
   RUNG wire#w1
      Contact( #Door2 )
   END_RUNG wire#w3
   RUNG wire#w3
      Move(in := 0, out1 => #SearchArea_Status)
   END_RUNG
   RUNG wire#w3
      S_Coil( #Error.WrongSequence2 )
   END_RUNG
   // the same network as SCL:
   #_w1 := (#"Step" = 2) AND (#SearchArea_Status = 1) AND NOT #Error.All AND #"E-Stop" AND #Door1;
   IF #_w1 AND NOT #SB1 AND NOT #SB2 AND NOT #Door2 THEN
       #"Step" := 0;
       #SearchArea_Status := 2;
   END_IF;
   IF #_w1 AND (#SB1 OR #SB2 OR #Door2) THEN
       #"Step" := 0;
       #SearchArea_Status := 0;
       #Error.WrongSequence2 := TRUE;
   END_IF;
END_REGION

REGION Network 8: 门2关闭
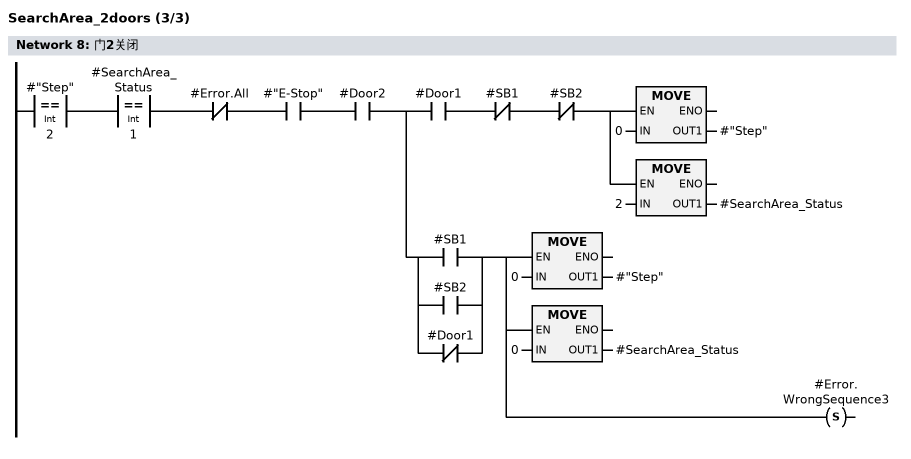
   RUNG wire#powerrail
      { S7_Templates := "SrcType := Int" } EQ_Contact(in1 := #"Step", in2 := 2)
      { S7_Templates := "SrcType := Int" } EQ_Contact(in1 := #SearchArea_Status, in2 := 1)
      I_Contact( #Error.All )
      Contact( #"E-Stop" )
      Contact( #Door2 )
      wire#w1
      Contact( #Door1 )
      I_Contact( #SB1 )
      I_Contact( #SB2 )
      wire#w2
      Move(in := 0, out1 => #"Step")
   END_RUNG
   RUNG wire#w2
      Move(in := 2, out1 => #SearchArea_Status)
   END_RUNG
   RUNG wire#w1
      Contact( #SB1 )
      wire#w3
      Move(in := 0, out1 => #"Step")
   END_RUNG
   RUNG wire#w1
      Contact( #SB2 )
   END_RUNG wire#w3
   RUNG wire#w1
      I_Contact( #Door1 )
   END_RUNG wire#w3
   RUNG wire#w3
      Move(in := 0, out1 => #SearchArea_Status)
   END_RUNG
   RUNG wire#w3
      S_Coil( #Error.WrongSequence3 )
   END_RUNG
   // the same network as SCL:
   #_w1 := (#"Step" = 2) AND (#SearchArea_Status = 1) AND NOT #Error.All AND #"E-Stop" AND #Door2;
   IF #_w1 AND #Door1 AND NOT #SB1 AND NOT #SB2 THEN
       #"Step" := 0;
       #SearchArea_Status := 2;
   END_IF;
   IF #_w1 AND (#SB1 OR #SB2 OR NOT #Door1) THEN
       #"Step" := 0;
       #SearchArea_Status := 0;
       #Error.WrongSequence3 := TRUE;
   END_IF;
END_REGION
END_FUNCTION_BLOCK

FUNCTION_BLOCK "FS_ACC"   // FB4, F_LAD
{ S7_Optimized_Access := 'TRUE' }
VERSION : 0.1
// stored: AutoNumber false, IsIECCheckEnabled false, UDAEnableTagReadback false
   VAR_INPUT
      ACK : Bool;
   END_VAR
   VAR_OUTPUT
      ES_OK : Bool;
   END_VAR
   VAR
      EStop1 { S7_SetPoint := 'True'} : ESTOP1;
      EStop2 { S7_SetPoint := 'True'} : ESTOP1;
      EStop3 { S7_SetPoint := 'True'} : ESTOP1;
      EStop4 { S7_SetPoint := 'True'} : ESTOP1;
      door1 : SFDOOR;
      door2 : SFDOOR;
      Key : SFDOOR;
      KeyControl : SFDOOR;
   END_VAR
BEGIN

REGION Network 1: E-Stop1
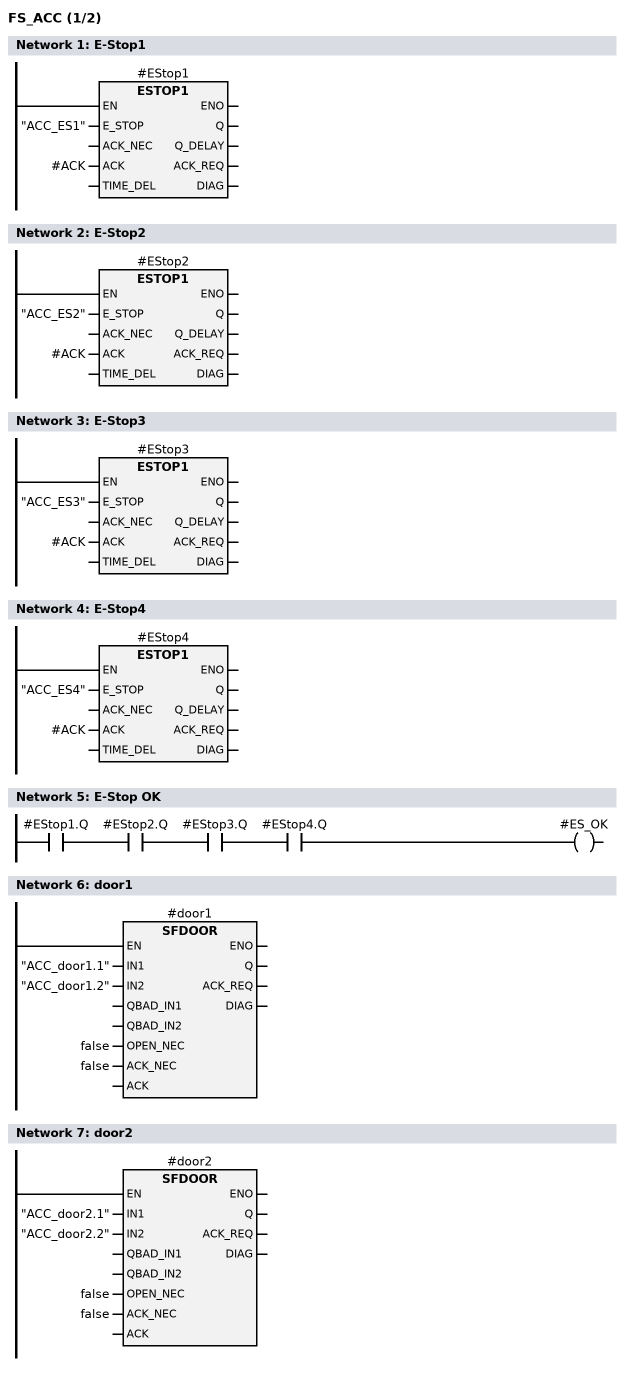
   RUNG wire#powerrail
      #EStop1.ESTOP1(E_STOP := "ACC_ES1", ACK_NEC :=, ACK := #ACK, TIME_DEL :=, Q =>, Q_DELAY =>, ACK_REQ =>, DIAG =>)
   END_RUNG
   // the same network as SCL:
   #EStop1(E_STOP := "ACC_ES1", ACK := #ACK);   // ESTOP1
END_REGION

REGION Network 2: E-Stop2
   RUNG wire#powerrail
      #EStop2.ESTOP1(E_STOP := "ACC_ES2", ACK_NEC :=, ACK := #ACK, TIME_DEL :=, Q =>, Q_DELAY =>, ACK_REQ =>, DIAG =>)
   END_RUNG
   // the same network as SCL:
   #EStop2(E_STOP := "ACC_ES2", ACK := #ACK);   // ESTOP1
END_REGION

REGION Network 3: E-Stop3
   RUNG wire#powerrail
      #EStop3.ESTOP1(E_STOP := "ACC_ES3", ACK_NEC :=, ACK := #ACK, TIME_DEL :=, Q =>, Q_DELAY =>, ACK_REQ =>, DIAG =>)
   END_RUNG
   // the same network as SCL:
   #EStop3(E_STOP := "ACC_ES3", ACK := #ACK);   // ESTOP1
END_REGION

REGION Network 4: E-Stop4
   RUNG wire#powerrail
      #EStop4.ESTOP1(E_STOP := "ACC_ES4", ACK_NEC :=, ACK := #ACK, TIME_DEL :=, Q =>, Q_DELAY =>, ACK_REQ =>, DIAG =>)
   END_RUNG
   // the same network as SCL:
   #EStop4(E_STOP := "ACC_ES4", ACK := #ACK);   // ESTOP1
END_REGION

REGION Network 5: E-Stop OK
   RUNG wire#powerrail
      Contact( #EStop1.Q )
      Contact( #EStop2.Q )
      Contact( #EStop3.Q )
      Contact( #EStop4.Q )
      Coil( #ES_OK )
   END_RUNG
   // the same network as SCL:
   #ES_OK := #EStop1.Q AND #EStop2.Q AND #EStop3.Q AND #EStop4.Q;
END_REGION

REGION Network 6: door1
   RUNG wire#powerrail
      #door1.SFDOOR(IN1 := "ACC_door1.1", IN2 := "ACC_door1.2", QBAD_IN1 :=, QBAD_IN2 :=, OPEN_NEC := false, ACK_NEC := false, ACK :=, Q =>, ACK_REQ =>, DIAG =>)
   END_RUNG
   // the same network as SCL:
   #door1(IN1 := "ACC_door1.1", IN2 := "ACC_door1.2", OPEN_NEC := false, ACK_NEC := false);   // SFDOOR
END_REGION

REGION Network 7: door2
   RUNG wire#powerrail
      #door2.SFDOOR(IN1 := "ACC_door2.1", IN2 := "ACC_door2.2", QBAD_IN1 :=, QBAD_IN2 :=, OPEN_NEC := false, ACK_NEC := false, ACK :=, Q =>, ACK_REQ =>, DIAG =>)
   END_RUNG
   // the same network as SCL:
   #door2(IN1 := "ACC_door2.1", IN2 := "ACC_door2.2", OPEN_NEC := false, ACK_NEC := false);   // SFDOOR
END_REGION

REGION Network 8: Key
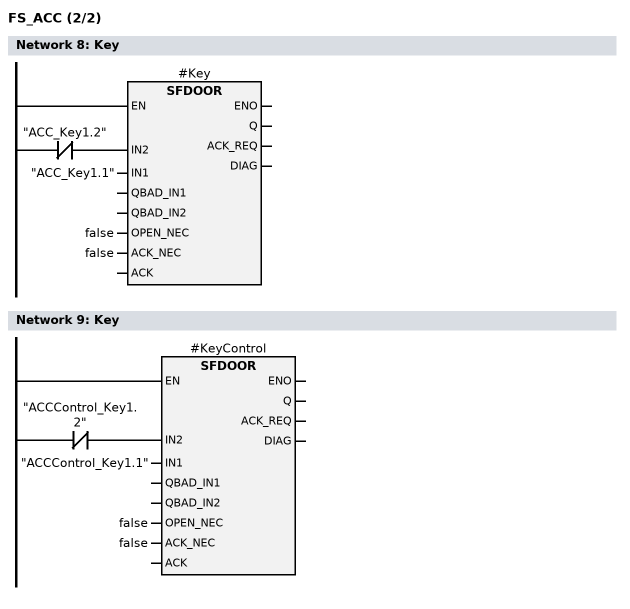
   RUNG wire#powerrail
      #Key.SFDOOR(IN2 := wire#w1, IN1 := "ACC_Key1.1", QBAD_IN1 :=, QBAD_IN2 :=, OPEN_NEC := false, ACK_NEC := false, ACK :=, Q =>, ACK_REQ =>, DIAG =>)
   END_RUNG
   RUNG wire#powerrail
      I_Contact( "ACC_Key1.2" )
   END_RUNG wire#w1
   // the same network as SCL:
   #Key(IN2 := NOT "ACC_Key1.2", IN1 := "ACC_Key1.1", OPEN_NEC := false, ACK_NEC := false);   // SFDOOR
END_REGION

REGION Network 9: Key
   RUNG wire#powerrail
      #KeyControl.SFDOOR(IN2 := wire#w1, IN1 := "ACCControl_Key1.1", QBAD_IN1 :=, QBAD_IN2 :=, OPEN_NEC := false, ACK_NEC := false, ACK :=, Q =>, ACK_REQ =>, DIAG =>)
   END_RUNG
   RUNG wire#powerrail
      I_Contact( "ACCControl_Key1.2" )
   END_RUNG wire#w1
   // the same network as SCL:
   #KeyControl(IN2 := NOT "ACCControl_Key1.2", IN1 := "ACCControl_Key1.1", OPEN_NEC := false, ACK_NEC := false);   // SFDOOR
END_REGION
END_FUNCTION_BLOCK

FUNCTION_BLOCK "FS_Room1"   // FB2, F_LAD
{ S7_Optimized_Access := 'TRUE' }
VERSION : 0.1
// 急停：2NC 硬件组态配置
// 1,急停故障
// 2,急停已恢复，需要确认
// 
// 
// 钥匙：1NC+1NO
// 1，钥匙电磁基座信号不匹配
// 2，基座信号正常，需要确认
// 3，安全钥匙2个电磁基座信号一致性故障，均显示插入
// 4，安全钥匙2个电磁基座信号一致性正常，需要确认
// 
// 门：2NC时关闭
// 1，门信号不一致，需要同时开同时关闭
// stored: AutoNumber true, IsIECCheckEnabled false, UDAEnableTagReadback false
   VAR_INPUT
      ACK : Bool;
   END_VAR
   VAR_OUTPUT
      ES_OK : Bool;
   END_VAR
   VAR
      EStop1 { S7_SetPoint := 'True'} : ESTOP1;
      EStop2 { S7_SetPoint := 'True'} : ESTOP1;
      EStop3 { S7_SetPoint := 'True'} : ESTOP1;
      EStop4 { S7_SetPoint := 'True'} : ESTOP1;
      EStop5 { S7_SetPoint := 'True'} : ESTOP1;
      EStop6 : ESTOP1;
      door : SFDOOR;
      Key : SFDOOR;
      KeyControl : SFDOOR;
      Door_Timer : TON;
      Key1 : TON;
      KeyControl1 : TON;
      Key_InDoor : Bool;
      Key_InControl : Bool;
   END_VAR
BEGIN

REGION Network 1: E-Stop1
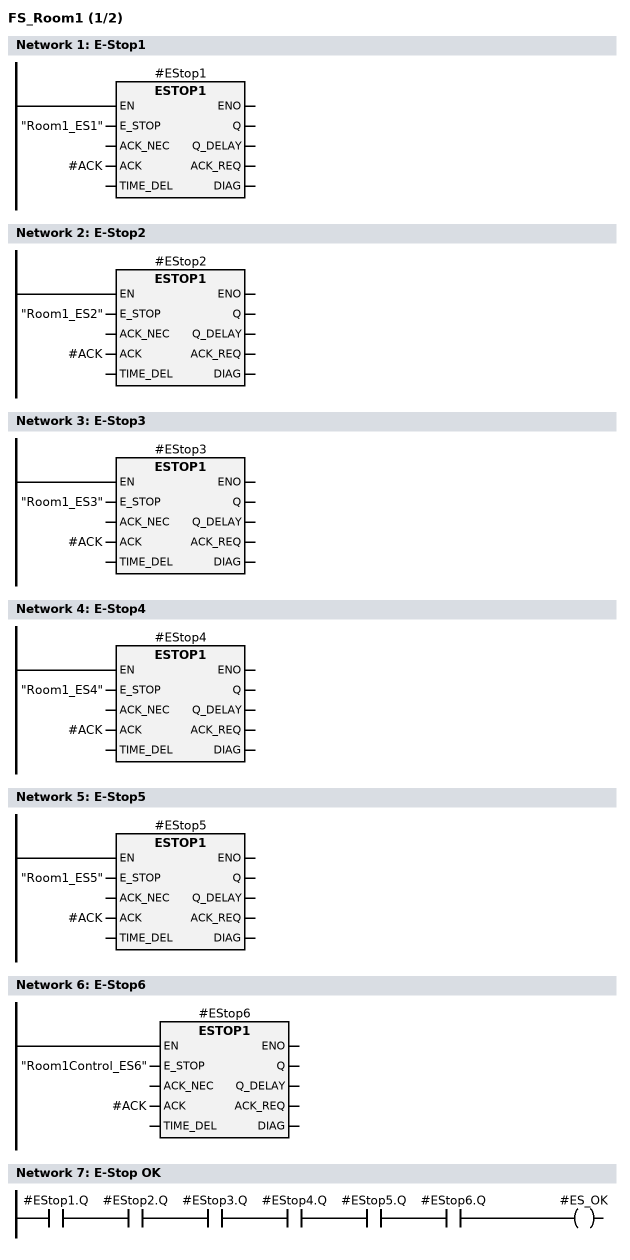
   RUNG wire#powerrail
      #EStop1.ESTOP1(E_STOP := "Room1_ES1", ACK_NEC :=, ACK := #ACK, TIME_DEL :=, Q =>, Q_DELAY =>, ACK_REQ =>, DIAG =>)
   END_RUNG
   // the same network as SCL:
   #EStop1(E_STOP := "Room1_ES1", ACK := #ACK);   // ESTOP1
END_REGION

REGION Network 2: E-Stop2
   RUNG wire#powerrail
      #EStop2.ESTOP1(E_STOP := "Room1_ES2", ACK_NEC :=, ACK := #ACK, TIME_DEL :=, Q =>, Q_DELAY =>, ACK_REQ =>, DIAG =>)
   END_RUNG
   // the same network as SCL:
   #EStop2(E_STOP := "Room1_ES2", ACK := #ACK);   // ESTOP1
END_REGION

REGION Network 3: E-Stop3
   RUNG wire#powerrail
      #EStop3.ESTOP1(E_STOP := "Room1_ES3", ACK_NEC :=, ACK := #ACK, TIME_DEL :=, Q =>, Q_DELAY =>, ACK_REQ =>, DIAG =>)
   END_RUNG
   // the same network as SCL:
   #EStop3(E_STOP := "Room1_ES3", ACK := #ACK);   // ESTOP1
END_REGION

REGION Network 4: E-Stop4
   RUNG wire#powerrail
      #EStop4.ESTOP1(E_STOP := "Room1_ES4", ACK_NEC :=, ACK := #ACK, TIME_DEL :=, Q =>, Q_DELAY =>, ACK_REQ =>, DIAG =>)
   END_RUNG
   // the same network as SCL:
   #EStop4(E_STOP := "Room1_ES4", ACK := #ACK);   // ESTOP1
END_REGION

REGION Network 5: E-Stop5
   RUNG wire#powerrail
      #EStop5.ESTOP1(E_STOP := "Room1_ES5", ACK_NEC :=, ACK := #ACK, TIME_DEL :=, Q =>, Q_DELAY =>, ACK_REQ =>, DIAG =>)
   END_RUNG
   // the same network as SCL:
   #EStop5(E_STOP := "Room1_ES5", ACK := #ACK);   // ESTOP1
END_REGION

REGION Network 6: E-Stop6
   RUNG wire#powerrail
      #EStop6.ESTOP1(E_STOP := "Room1Control_ES6", ACK_NEC :=, ACK := #ACK, TIME_DEL :=, Q =>, Q_DELAY =>, ACK_REQ =>, DIAG =>)
   END_RUNG
   // the same network as SCL:
   #EStop6(E_STOP := "Room1Control_ES6", ACK := #ACK);   // ESTOP1
END_REGION

REGION Network 7: E-Stop OK
   RUNG wire#powerrail
      Contact( #EStop1.Q )
      Contact( #EStop2.Q )
      Contact( #EStop3.Q )
      Contact( #EStop4.Q )
      Contact( #EStop5.Q )
      Contact( #EStop6.Q )
      Coil( #ES_OK )
   END_RUNG
   // the same network as SCL:
   #ES_OK := #EStop1.Q AND #EStop2.Q AND #EStop3.Q AND #EStop4.Q AND #EStop5.Q AND #EStop6.Q;
END_REGION

REGION Network 8: door
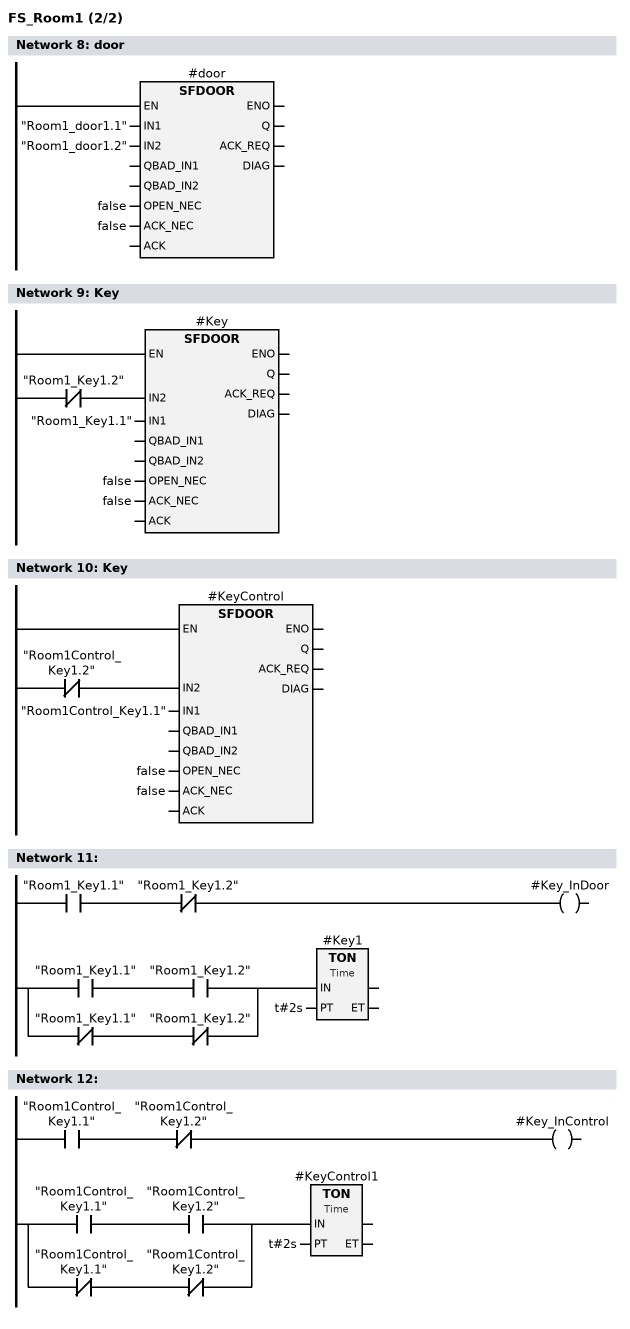
   RUNG wire#powerrail
      #door.SFDOOR(IN1 := "Room1_door1.1", IN2 := "Room1_door1.2", QBAD_IN1 :=, QBAD_IN2 :=, OPEN_NEC := false, ACK_NEC := false, ACK :=, Q =>, ACK_REQ =>, DIAG =>)
   END_RUNG
   // the same network as SCL:
   #door(IN1 := "Room1_door1.1", IN2 := "Room1_door1.2", OPEN_NEC := false, ACK_NEC := false);   // SFDOOR
END_REGION

REGION Network 9: Key
   RUNG wire#powerrail
      #Key.SFDOOR(IN2 := wire#w1, IN1 := "Room1_Key1.1", QBAD_IN1 :=, QBAD_IN2 :=, OPEN_NEC := false, ACK_NEC := false, ACK :=, Q =>, ACK_REQ =>, DIAG =>)
   END_RUNG
   RUNG wire#powerrail
      I_Contact( "Room1_Key1.2" )
   END_RUNG wire#w1
   // the same network as SCL:
   #Key(IN2 := NOT "Room1_Key1.2", IN1 := "Room1_Key1.1", OPEN_NEC := false, ACK_NEC := false);   // SFDOOR
END_REGION

REGION Network 10: Key
   RUNG wire#powerrail
      #KeyControl.SFDOOR(IN2 := wire#w1, IN1 := "Room1Control_Key1.1", QBAD_IN1 :=, QBAD_IN2 :=, OPEN_NEC := false, ACK_NEC := false, ACK :=, Q =>, ACK_REQ =>, DIAG =>)
   END_RUNG
   RUNG wire#powerrail
      I_Contact( "Room1Control_Key1.2" )
   END_RUNG wire#w1
   // the same network as SCL:
   #KeyControl(IN2 := NOT "Room1Control_Key1.2",   // SFDOOR
               IN1 := "Room1Control_Key1.1",
               OPEN_NEC := false,
               ACK_NEC := false);
END_REGION

REGION Network 11
   RUNG wire#powerrail
      Contact( "Room1_Key1.1" )
      I_Contact( "Room1_Key1.2" )
      Coil( #Key_InDoor )
   END_RUNG
   RUNG wire#powerrail
      Contact( "Room1_Key1.1" )
      Contact( "Room1_Key1.2" )
      wire#w1
      { S7_Templates := "[time_type := Time, codedbool_type := DInt]" } #Key1.TON(pt := t#2s, et =>)
   END_RUNG
   RUNG wire#powerrail
      I_Contact( "Room1_Key1.1" )
      I_Contact( "Room1_Key1.2" )
   END_RUNG wire#w1
   // the same network as SCL:
   #Key_InDoor := "Room1_Key1.1" AND NOT "Room1_Key1.2";
   #Key1.TON(IN := ("Room1_Key1.1" AND "Room1_Key1.2") OR (NOT "Room1_Key1.1" AND NOT "Room1_Key1.2"),
             PT := t#2s);
END_REGION

REGION Network 12
   RUNG wire#powerrail
      Contact( "Room1Control_Key1.1" )
      I_Contact( "Room1Control_Key1.2" )
      Coil( #Key_InControl )
   END_RUNG
   RUNG wire#powerrail
      Contact( "Room1Control_Key1.1" )
      Contact( "Room1Control_Key1.2" )
      wire#w1
      { S7_Templates := "[time_type := Time, codedbool_type := DInt]" } #KeyControl1.TON(pt := t#2s, et =>)
   END_RUNG
   RUNG wire#powerrail
      I_Contact( "Room1Control_Key1.1" )
      I_Contact( "Room1Control_Key1.2" )
   END_RUNG wire#w1
   // the same network as SCL:
   #Key_InControl := "Room1Control_Key1.1" AND NOT "Room1Control_Key1.2";
   #KeyControl1.TON(IN := ("Room1Control_Key1.1" AND "Room1Control_Key1.2") OR (NOT "Room1Control_Key1.1" AND NOT "Room1Control_Key1.2"),
                    PT := t#2s);
END_REGION
END_FUNCTION_BLOCK

FUNCTION_BLOCK "FS_Room2"   // FB3, F_LAD
{ S7_Optimized_Access := 'TRUE' }
VERSION : 0.1
// stored: AutoNumber false, IsIECCheckEnabled false, UDAEnableTagReadback false
   VAR_INPUT
      ACK : Bool;
   END_VAR
   VAR_OUTPUT
      ES_OK : Bool;
   END_VAR
   VAR
      EStop1 { S7_SetPoint := 'True'} : ESTOP1;
      EStop2 { S7_SetPoint := 'True'} : ESTOP1;
      EStop3 { S7_SetPoint := 'True'} : ESTOP1;
      EStop4 { S7_SetPoint := 'True'} : ESTOP1;
      EStop5 { S7_SetPoint := 'True'} : ESTOP1;
      EStop6 : ESTOP1;
      door : SFDOOR;
      Key : SFDOOR;
      KeyControl : SFDOOR;
   END_VAR
BEGIN

REGION Network 1: E-Stop1
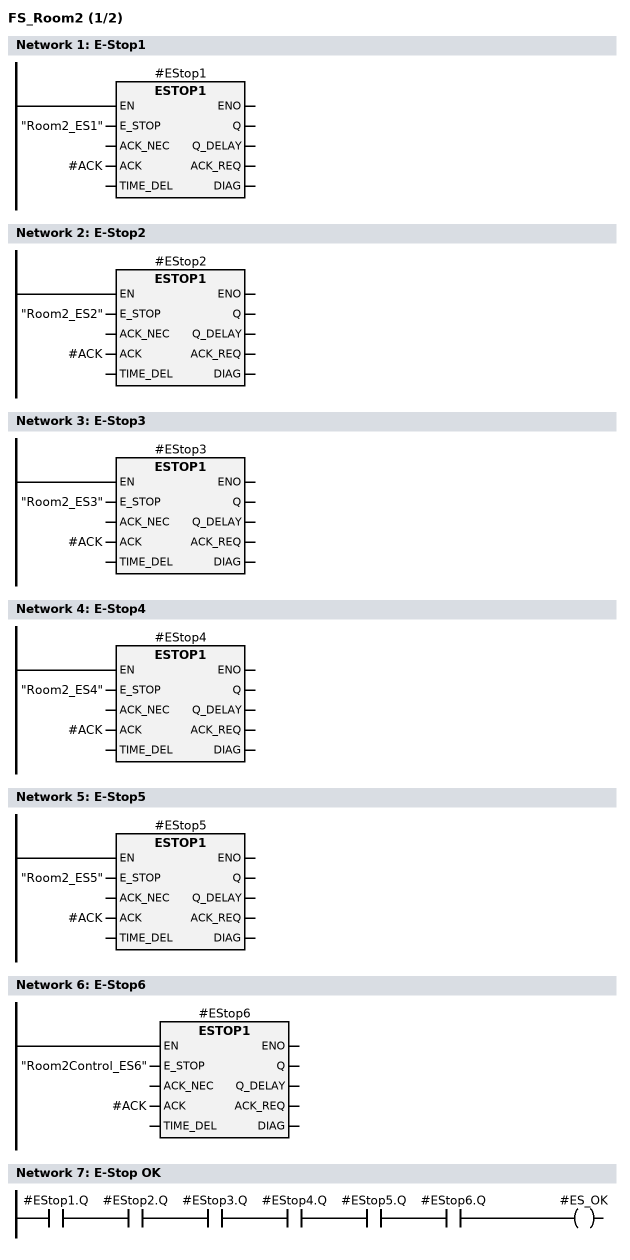
   RUNG wire#powerrail
      #EStop1.ESTOP1(E_STOP := "Room2_ES1", ACK_NEC :=, ACK := #ACK, TIME_DEL :=, Q =>, Q_DELAY =>, ACK_REQ =>, DIAG =>)
   END_RUNG
   // the same network as SCL:
   #EStop1(E_STOP := "Room2_ES1", ACK := #ACK);   // ESTOP1
END_REGION

REGION Network 2: E-Stop2
   RUNG wire#powerrail
      #EStop2.ESTOP1(E_STOP := "Room2_ES2", ACK_NEC :=, ACK := #ACK, TIME_DEL :=, Q =>, Q_DELAY =>, ACK_REQ =>, DIAG =>)
   END_RUNG
   // the same network as SCL:
   #EStop2(E_STOP := "Room2_ES2", ACK := #ACK);   // ESTOP1
END_REGION

REGION Network 3: E-Stop3
   RUNG wire#powerrail
      #EStop3.ESTOP1(E_STOP := "Room2_ES3", ACK_NEC :=, ACK := #ACK, TIME_DEL :=, Q =>, Q_DELAY =>, ACK_REQ =>, DIAG =>)
   END_RUNG
   // the same network as SCL:
   #EStop3(E_STOP := "Room2_ES3", ACK := #ACK);   // ESTOP1
END_REGION

REGION Network 4: E-Stop4
   RUNG wire#powerrail
      #EStop4.ESTOP1(E_STOP := "Room2_ES4", ACK_NEC :=, ACK := #ACK, TIME_DEL :=, Q =>, Q_DELAY =>, ACK_REQ =>, DIAG =>)
   END_RUNG
   // the same network as SCL:
   #EStop4(E_STOP := "Room2_ES4", ACK := #ACK);   // ESTOP1
END_REGION

REGION Network 5: E-Stop5
   RUNG wire#powerrail
      #EStop5.ESTOP1(E_STOP := "Room2_ES5", ACK_NEC :=, ACK := #ACK, TIME_DEL :=, Q =>, Q_DELAY =>, ACK_REQ =>, DIAG =>)
   END_RUNG
   // the same network as SCL:
   #EStop5(E_STOP := "Room2_ES5", ACK := #ACK);   // ESTOP1
END_REGION

REGION Network 6: E-Stop6
   RUNG wire#powerrail
      #EStop6.ESTOP1(E_STOP := "Room2Control_ES6", ACK_NEC :=, ACK := #ACK, TIME_DEL :=, Q =>, Q_DELAY =>, ACK_REQ =>, DIAG =>)
   END_RUNG
   // the same network as SCL:
   #EStop6(E_STOP := "Room2Control_ES6", ACK := #ACK);   // ESTOP1
END_REGION

REGION Network 7: E-Stop OK
   RUNG wire#powerrail
      Contact( #EStop1.Q )
      Contact( #EStop2.Q )
      Contact( #EStop3.Q )
      Contact( #EStop4.Q )
      Contact( #EStop5.Q )
      Contact( #EStop6.Q )
      Coil( #ES_OK )
   END_RUNG
   // the same network as SCL:
   #ES_OK := #EStop1.Q AND #EStop2.Q AND #EStop3.Q AND #EStop4.Q AND #EStop5.Q AND #EStop6.Q;
END_REGION

REGION Network 8: door
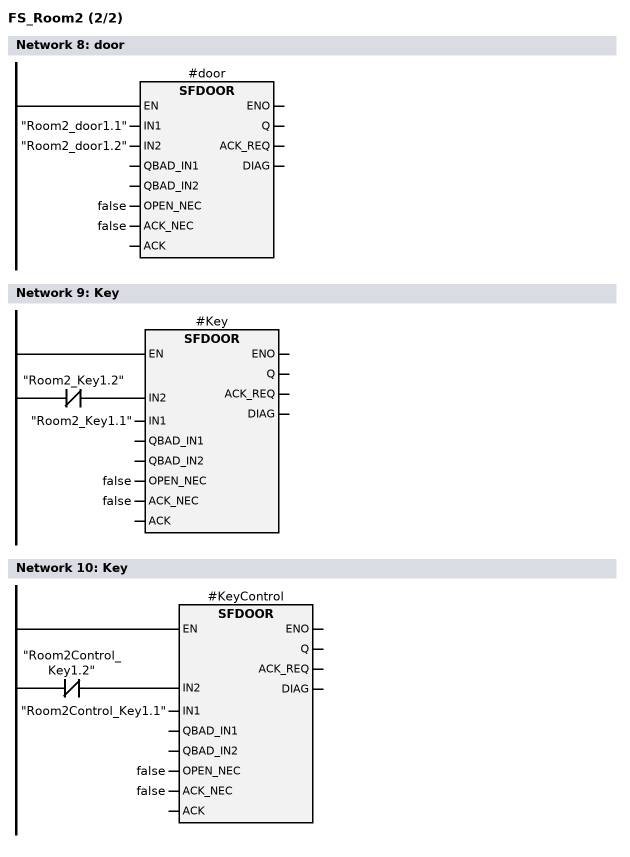
   RUNG wire#powerrail
      #door.SFDOOR(IN1 := "Room2_door1.1", IN2 := "Room2_door1.2", QBAD_IN1 :=, QBAD_IN2 :=, OPEN_NEC := false, ACK_NEC := false, ACK :=, Q =>, ACK_REQ =>, DIAG =>)
   END_RUNG
   // the same network as SCL:
   #door(IN1 := "Room2_door1.1", IN2 := "Room2_door1.2", OPEN_NEC := false, ACK_NEC := false);   // SFDOOR
END_REGION

REGION Network 9: Key
   RUNG wire#powerrail
      #Key.SFDOOR(IN2 := wire#w1, IN1 := "Room2_Key1.1", QBAD_IN1 :=, QBAD_IN2 :=, OPEN_NEC := false, ACK_NEC := false, ACK :=, Q =>, ACK_REQ =>, DIAG =>)
   END_RUNG
   RUNG wire#powerrail
      I_Contact( "Room2_Key1.2" )
   END_RUNG wire#w1
   // the same network as SCL:
   #Key(IN2 := NOT "Room2_Key1.2", IN1 := "Room2_Key1.1", OPEN_NEC := false, ACK_NEC := false);   // SFDOOR
END_REGION

REGION Network 10: Key
   RUNG wire#powerrail
      #KeyControl.SFDOOR(IN2 := wire#w1, IN1 := "Room2Control_Key1.1", QBAD_IN1 :=, QBAD_IN2 :=, OPEN_NEC := false, ACK_NEC := false, ACK :=, Q =>, ACK_REQ =>, DIAG =>)
   END_RUNG
   RUNG wire#powerrail
      I_Contact( "Room2Control_Key1.2" )
   END_RUNG wire#w1
   // the same network as SCL:
   #KeyControl(IN2 := NOT "Room2Control_Key1.2",   // SFDOOR
               IN1 := "Room2Control_Key1.1",
               OPEN_NEC := false,
               ACK_NEC := false);
END_REGION
END_FUNCTION_BLOCK

FUNCTION_BLOCK "FS_VerticalBeam"   // FB5, F_LAD
{ S7_Optimized_Access := 'TRUE' }
VERSION : 0.1
// stored: AutoNumber false, IsIECCheckEnabled false, UDAEnableTagReadback false
   VAR_INPUT
      ACK : Bool;
   END_VAR
   VAR_OUTPUT
      ES_OK : Bool;
   END_VAR
   VAR
      EStop1 { S7_SetPoint := 'True'} : ESTOP1;
      EStop2 { S7_SetPoint := 'True'} : ESTOP1;
      EStop3 { S7_SetPoint := 'True'} : ESTOP1;
      EStop4 { S7_SetPoint := 'True'} : ESTOP1;
      door1 : SFDOOR;
      door2 : SFDOOR;
      Key : SFDOOR;
      KeyControl : SFDOOR;
   END_VAR
BEGIN

REGION Network 1: E-Stop1
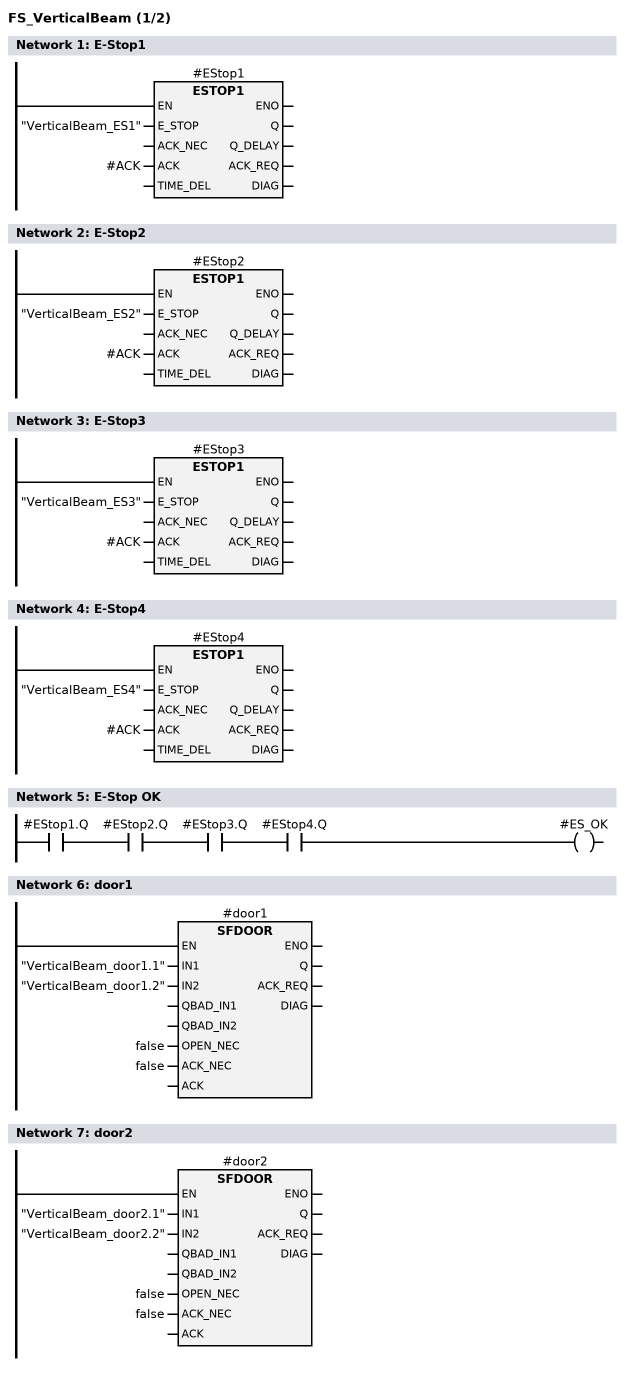
   RUNG wire#powerrail
      #EStop1.ESTOP1(E_STOP := "VerticalBeam_ES1", ACK_NEC :=, ACK := #ACK, TIME_DEL :=, Q =>, Q_DELAY =>, ACK_REQ =>, DIAG =>)
   END_RUNG
   // the same network as SCL:
   #EStop1(E_STOP := "VerticalBeam_ES1", ACK := #ACK);   // ESTOP1
END_REGION

REGION Network 2: E-Stop2
   RUNG wire#powerrail
      #EStop2.ESTOP1(E_STOP := "VerticalBeam_ES2", ACK_NEC :=, ACK := #ACK, TIME_DEL :=, Q =>, Q_DELAY =>, ACK_REQ =>, DIAG =>)
   END_RUNG
   // the same network as SCL:
   #EStop2(E_STOP := "VerticalBeam_ES2", ACK := #ACK);   // ESTOP1
END_REGION

REGION Network 3: E-Stop3
   RUNG wire#powerrail
      #EStop3.ESTOP1(E_STOP := "VerticalBeam_ES3", ACK_NEC :=, ACK := #ACK, TIME_DEL :=, Q =>, Q_DELAY =>, ACK_REQ =>, DIAG =>)
   END_RUNG
   // the same network as SCL:
   #EStop3(E_STOP := "VerticalBeam_ES3", ACK := #ACK);   // ESTOP1
END_REGION

REGION Network 4: E-Stop4
   RUNG wire#powerrail
      #EStop4.ESTOP1(E_STOP := "VerticalBeam_ES4", ACK_NEC :=, ACK := #ACK, TIME_DEL :=, Q =>, Q_DELAY =>, ACK_REQ =>, DIAG =>)
   END_RUNG
   // the same network as SCL:
   #EStop4(E_STOP := "VerticalBeam_ES4", ACK := #ACK);   // ESTOP1
END_REGION

REGION Network 5: E-Stop OK
   RUNG wire#powerrail
      Contact( #EStop1.Q )
      Contact( #EStop2.Q )
      Contact( #EStop3.Q )
      Contact( #EStop4.Q )
      Coil( #ES_OK )
   END_RUNG
   // the same network as SCL:
   #ES_OK := #EStop1.Q AND #EStop2.Q AND #EStop3.Q AND #EStop4.Q;
END_REGION

REGION Network 6: door1
   RUNG wire#powerrail
      #door1.SFDOOR(IN1 := "VerticalBeam_door1.1", IN2 := "VerticalBeam_door1.2", QBAD_IN1 :=, QBAD_IN2 :=, OPEN_NEC := false, ACK_NEC := false, ACK :=, Q =>, ACK_REQ =>, DIAG =>)
   END_RUNG
   // the same network as SCL:
   #door1(IN1 := "VerticalBeam_door1.1", IN2 := "VerticalBeam_door1.2", OPEN_NEC := false, ACK_NEC := false);   // SFDOOR
END_REGION

REGION Network 7: door2
   RUNG wire#powerrail
      #door2.SFDOOR(IN1 := "VerticalBeam_door2.1", IN2 := "VerticalBeam_door2.2", QBAD_IN1 :=, QBAD_IN2 :=, OPEN_NEC := false, ACK_NEC := false, ACK :=, Q =>, ACK_REQ =>, DIAG =>)
   END_RUNG
   // the same network as SCL:
   #door2(IN1 := "VerticalBeam_door2.1", IN2 := "VerticalBeam_door2.2", OPEN_NEC := false, ACK_NEC := false);   // SFDOOR
END_REGION

REGION Network 8: Key
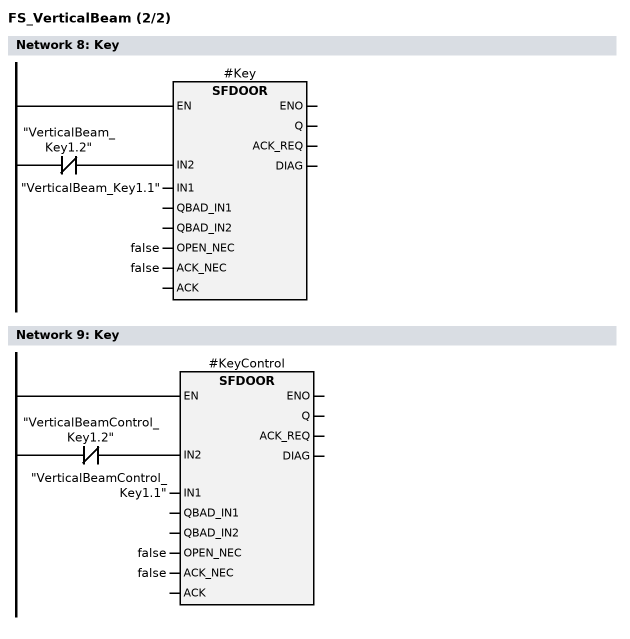
   RUNG wire#powerrail
      #Key.SFDOOR(IN2 := wire#w1, IN1 := "VerticalBeam_Key1.1", QBAD_IN1 :=, QBAD_IN2 :=, OPEN_NEC := false, ACK_NEC := false, ACK :=, Q =>, ACK_REQ =>, DIAG =>)
   END_RUNG
   RUNG wire#powerrail
      I_Contact( "VerticalBeam_Key1.2" )
   END_RUNG wire#w1
   // the same network as SCL:
   #Key(IN2 := NOT "VerticalBeam_Key1.2", IN1 := "VerticalBeam_Key1.1", OPEN_NEC := false, ACK_NEC := false);   // SFDOOR
END_REGION

REGION Network 9: Key
   RUNG wire#powerrail
      #KeyControl.SFDOOR(IN2 := wire#w1, IN1 := "VerticalBeamControl_Key1.1", QBAD_IN1 :=, QBAD_IN2 :=, OPEN_NEC := false, ACK_NEC := false, ACK :=, Q =>, ACK_REQ =>, DIAG =>)
   END_RUNG
   RUNG wire#powerrail
      I_Contact( "VerticalBeamControl_Key1.2" )
   END_RUNG wire#w1
   // the same network as SCL:
   #KeyControl(IN2 := NOT "VerticalBeamControl_Key1.2",   // SFDOOR
               IN1 := "VerticalBeamControl_Key1.1",
               OPEN_NEC := false,
               ACK_NEC := false);
END_REGION
END_FUNCTION_BLOCK

FUNCTION "F_ChannelDia" : Void   // FC2, F_LAD
{ S7_Optimized_Access := 'TRUE' }
VERSION : 0.1
// stored: AutoNumber true, IsIECCheckEnabled false, UDAEnableTagReadback false
   VAR_INPUT
      PASS_OUT : Bool;
      QBAD : Bool;
      ACK_REQ : Bool;
      Channel0_ValueStatus : Bool;
      Channel1_ValueStatus : Bool;
      Channel2_ValueStatus : Bool;
      Channel3_ValueStatus : Bool;
      Channel4_ValueStatus : Bool;
      Channel5_ValueStatus : Bool;
      Channel6_ValueStatus : Bool;
      Channel7_ValueStatus : Bool;
   END_VAR
   VAR_OUTPUT
      FIODia : "FIODia";
   END_VAR
   VAR_TEMP   // added for the SCL form of the ladder/FBD networks
      _w1 : Bool;
   END_VAR
BEGIN

REGION Network 1: 模块钝化
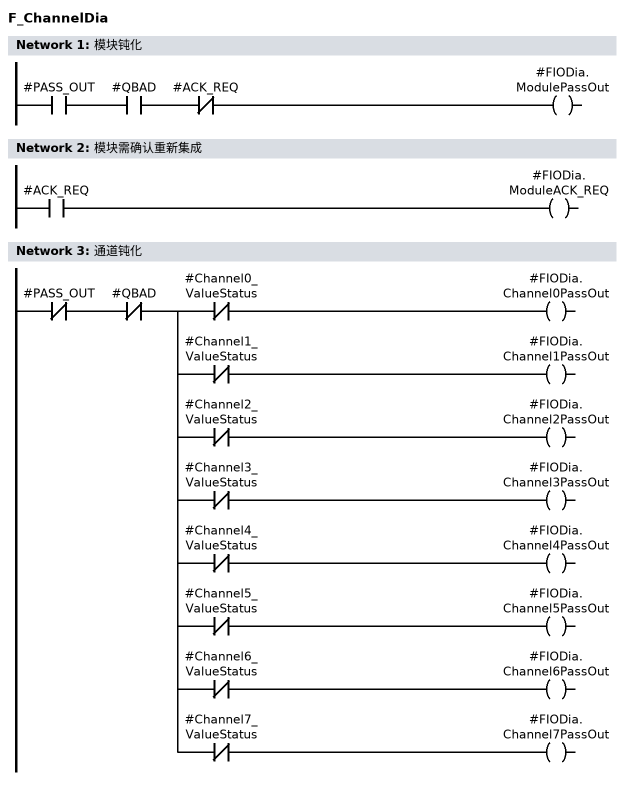
   RUNG wire#powerrail
      Contact( #PASS_OUT )
      Contact( #QBAD )
      I_Contact( #ACK_REQ )
      Coil( #FIODia.ModulePassOut )
   END_RUNG
   // the same network as SCL:
   #FIODia.ModulePassOut := #PASS_OUT AND #QBAD AND NOT #ACK_REQ;
END_REGION

REGION Network 2: 模块需确认重新集成
   RUNG wire#powerrail
      Contact( #ACK_REQ )
      Coil( #FIODia.ModuleACK_REQ )
   END_RUNG
   // the same network as SCL:
   #FIODia.ModuleACK_REQ := #ACK_REQ;
END_REGION

REGION Network 3: 通道钝化
   RUNG wire#powerrail
      I_Contact( #PASS_OUT )
      I_Contact( #QBAD )
      wire#w1
      I_Contact( #Channel0_ValueStatus )
      Coil( #FIODia.Channel0PassOut )
   END_RUNG
   RUNG wire#w1
      I_Contact( #Channel1_ValueStatus )
      Coil( #FIODia.Channel1PassOut )
   END_RUNG
   RUNG wire#w1
      I_Contact( #Channel2_ValueStatus )
      Coil( #FIODia.Channel2PassOut )
   END_RUNG
   RUNG wire#w1
      I_Contact( #Channel3_ValueStatus )
      Coil( #FIODia.Channel3PassOut )
   END_RUNG
   RUNG wire#w1
      I_Contact( #Channel4_ValueStatus )
      Coil( #FIODia.Channel4PassOut )
   END_RUNG
   RUNG wire#w1
      I_Contact( #Channel5_ValueStatus )
      Coil( #FIODia.Channel5PassOut )
   END_RUNG
   RUNG wire#w1
      I_Contact( #Channel6_ValueStatus )
      Coil( #FIODia.Channel6PassOut )
   END_RUNG
   RUNG wire#w1
      I_Contact( #Channel7_ValueStatus )
      Coil( #FIODia.Channel7PassOut )
   END_RUNG
   // the same network as SCL:
   #_w1 := NOT #PASS_OUT AND NOT #QBAD;
   #FIODia.Channel0PassOut := #_w1 AND NOT #Channel0_ValueStatus;
   #FIODia.Channel1PassOut := #_w1 AND NOT #Channel1_ValueStatus;
   #FIODia.Channel2PassOut := #_w1 AND NOT #Channel2_ValueStatus;
   #FIODia.Channel3PassOut := #_w1 AND NOT #Channel3_ValueStatus;
   #FIODia.Channel4PassOut := #_w1 AND NOT #Channel4_ValueStatus;
   #FIODia.Channel5PassOut := #_w1 AND NOT #Channel5_ValueStatus;
   #FIODia.Channel6PassOut := #_w1 AND NOT #Channel6_ValueStatus;
   #FIODia.Channel7PassOut := #_w1 AND NOT #Channel7_ValueStatus;
END_REGION
END_FUNCTION

FUNCTION "Interlock" : Void   // FC1, F_LAD
{ S7_Optimized_Access := 'TRUE' }
VERSION : 0.1
// stored: AutoNumber true, IsIECCheckEnabled false, UDAEnableTagReadback false
   VAR_INPUT
      Room1_Interlock : Bool;
      Room2_Interlock : Bool;
      ACC_Interlock : Bool;
      VerticalBeam_Interlock : Bool;
      "E-stop" : Bool;
   END_VAR
BEGIN

REGION Network 1
   // 暂未考虑模块钝化和通道钝化情况
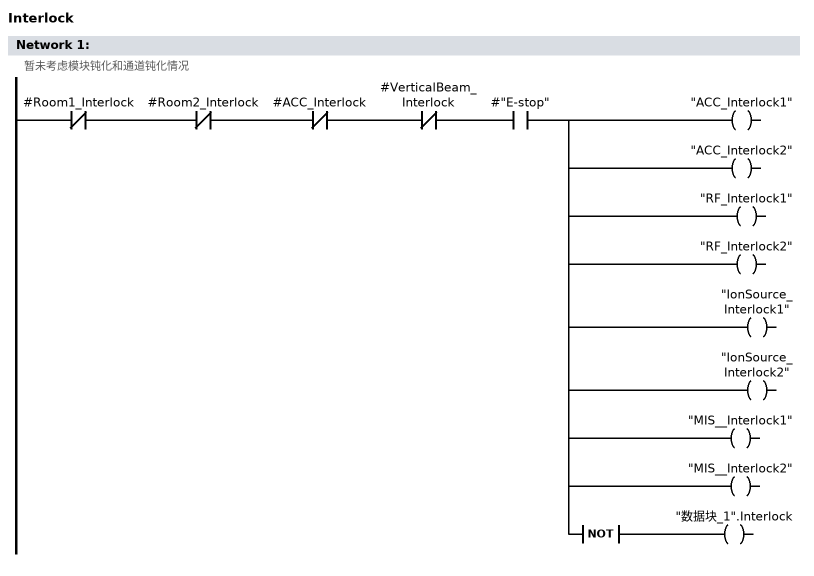
   RUNG wire#powerrail
      I_Contact( #Room1_Interlock )
      I_Contact( #Room2_Interlock )
      I_Contact( #ACC_Interlock )
      I_Contact( #VerticalBeam_Interlock )
      Contact( #"E-stop" )
      wire#w1
      Coil( "ACC_Interlock1" )
   END_RUNG
   RUNG wire#w1
      Coil( "ACC_Interlock2" )
   END_RUNG
   RUNG wire#w1
      Coil( "RF_Interlock1" )
   END_RUNG
   RUNG wire#w1
      Coil( "RF_Interlock2" )
   END_RUNG
   RUNG wire#w1
      Coil( "IonSource_Interlock1" )
   END_RUNG
   RUNG wire#w1
      Coil( "IonSource_Interlock2" )
   END_RUNG
   RUNG wire#w1
      Coil( "MIS__Interlock1" )
   END_RUNG
   RUNG wire#w1
      Coil( "MIS__Interlock2" )
   END_RUNG
   RUNG wire#w1
      Not()
      Coil( "数据块_1".Interlock )
   END_RUNG
   // the same network as SCL:
   "ACC_Interlock1" := NOT #Room1_Interlock AND NOT #Room2_Interlock AND NOT #ACC_Interlock AND NOT #VerticalBeam_Interlock AND #"E-stop";
   "ACC_Interlock2" := "ACC_Interlock1";
   "RF_Interlock1" := "ACC_Interlock1";
   "RF_Interlock2" := "ACC_Interlock1";
   "IonSource_Interlock1" := "ACC_Interlock1";
   "IonSource_Interlock2" := "ACC_Interlock1";
   "MIS__Interlock1" := "ACC_Interlock1";
   "MIS__Interlock2" := "ACC_Interlock1";
   "数据块_1".Interlock := NOT "ACC_Interlock1";
END_REGION
END_FUNCTION

FUNCTION_BLOCK "Main_Safety_RTG1"   // FB1, F_LAD
{ S7_Optimized_Access := 'TRUE' }
VERSION : 0.1
// stored: AutoNumber false, IsIECCheckEnabled false, UDAEnableTagReadback false
   VAR
      ACK_GL_Instance : ACK_GL;
      FS_Room1_Instance : "FS_Room1";
      FS_Room2_Instance : "FS_Room2";
      FS_ACC_Instance : "FS_ACC";
      FS_VerticalBeam_Instance : "FS_VerticalBeam";
   END_VAR
BEGIN

REGION Network 1: 全局确认钝化
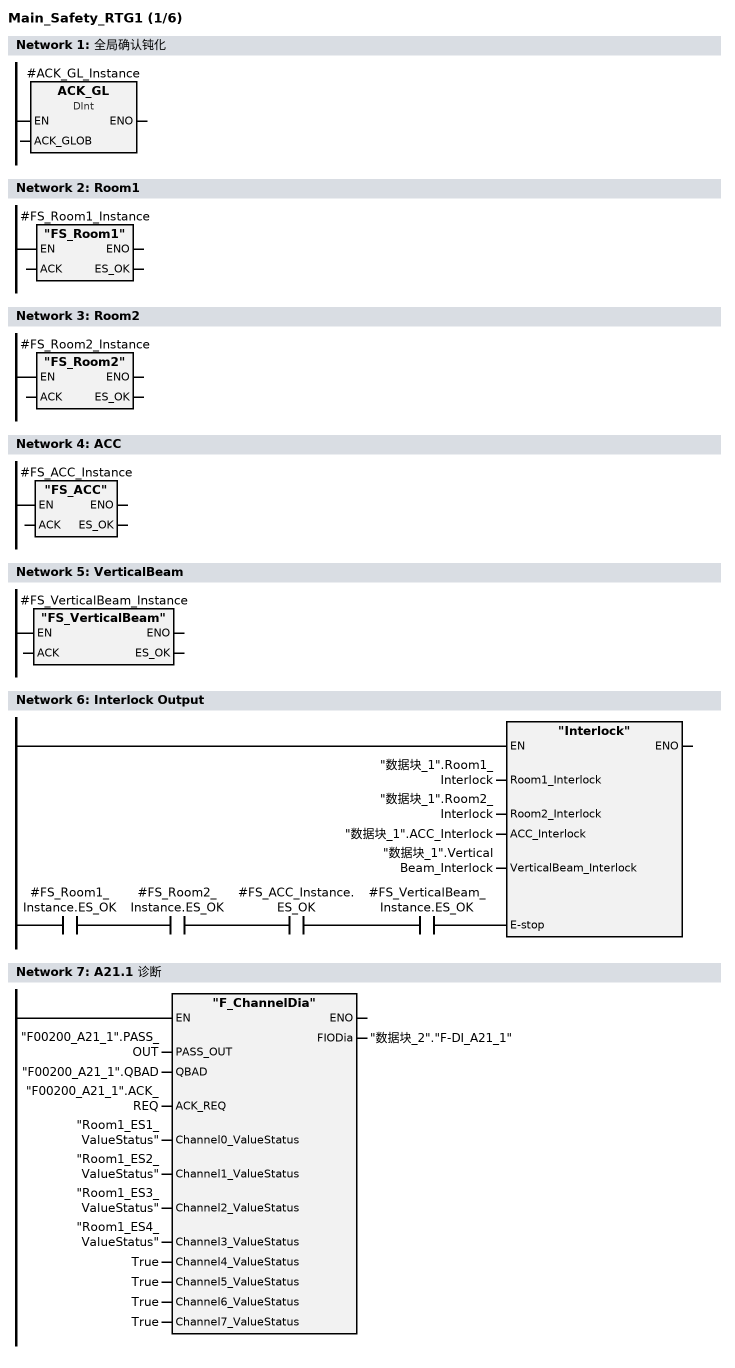
   RUNG wire#powerrail
      { S7_Templates := "codedbool_type := DInt" } #ACK_GL_Instance.ACK_GL(ACK_GLOB :=)
   END_RUNG
   // the same network as SCL:
   #ACK_GL_Instance();   // ACK_GL
END_REGION

REGION Network 2: Room1
   RUNG wire#powerrail
      #FS_Room1_Instance(ACK :=, ES_OK =>)
   END_RUNG
   // the same network as SCL:
   #FS_Room1_Instance();   // "FS_Room1"
END_REGION

REGION Network 3: Room2
   RUNG wire#powerrail
      #FS_Room2_Instance(ACK :=, ES_OK =>)
   END_RUNG
   // the same network as SCL:
   #FS_Room2_Instance();   // "FS_Room2"
END_REGION

REGION Network 4: ACC
   RUNG wire#powerrail
      #FS_ACC_Instance(ACK :=, ES_OK =>)
   END_RUNG
   // the same network as SCL:
   #FS_ACC_Instance();   // "FS_ACC"
END_REGION

REGION Network 5: VerticalBeam
   RUNG wire#powerrail
      #FS_VerticalBeam_Instance(ACK :=, ES_OK =>)
   END_RUNG
   // the same network as SCL:
   #FS_VerticalBeam_Instance();   // "FS_VerticalBeam"
END_REGION

REGION Network 6: Interlock Output
   RUNG wire#powerrail
      "Interlock"(Room1_Interlock := "数据块_1".Room1_Interlock, Room2_Interlock := "数据块_1".Room2_Interlock, ACC_Interlock := "数据块_1".ACC_Interlock, VerticalBeam_Interlock := "数据块_1".VerticalBeam_Interlock, "E-stop" := wire#w1)
   END_RUNG
   RUNG wire#powerrail
      Contact( #FS_Room1_Instance.ES_OK )
      Contact( #FS_Room2_Instance.ES_OK )
      Contact( #FS_ACC_Instance.ES_OK )
      Contact( #FS_VerticalBeam_Instance.ES_OK )
   END_RUNG wire#w1
   // the same network as SCL:
   "Interlock"(Room1_Interlock := "数据块_1".Room1_Interlock,
               Room2_Interlock := "数据块_1".Room2_Interlock,
               ACC_Interlock := "数据块_1".ACC_Interlock,
               VerticalBeam_Interlock := "数据块_1".VerticalBeam_Interlock,
               "E-stop" := #FS_Room1_Instance.ES_OK AND #FS_Room2_Instance.ES_OK AND #FS_ACC_Instance.ES_OK AND #FS_VerticalBeam_Instance.ES_OK);
END_REGION

REGION Network 7: A21.1 诊断
   RUNG wire#powerrail
      "F_ChannelDia"(PASS_OUT := "F00200_A21_1".PASS_OUT, QBAD := "F00200_A21_1".QBAD, ACK_REQ := "F00200_A21_1".ACK_REQ, Channel0_ValueStatus := "Room1_ES1_ValueStatus", Channel1_ValueStatus := "Room1_ES2_ValueStatus", Channel2_ValueStatus := "Room1_ES3_ValueStatus", Channel3_ValueStatus := "Room1_ES4_ValueStatus", Channel4_ValueStatus := True, Channel5_ValueStatus := True, Channel6_ValueStatus := True, Channel7_ValueStatus := True, FIODia => "数据块_2"."F-DI_A21_1")
   END_RUNG
   // the same network as SCL:
   "F_ChannelDia"(PASS_OUT := "F00200_A21_1".PASS_OUT,
                  QBAD := "F00200_A21_1".QBAD,
                  ACK_REQ := "F00200_A21_1".ACK_REQ,
                  Channel0_ValueStatus := "Room1_ES1_ValueStatus",
                  Channel1_ValueStatus := "Room1_ES2_ValueStatus",
                  Channel2_ValueStatus := "Room1_ES3_ValueStatus",
                  Channel3_ValueStatus := "Room1_ES4_ValueStatus",
                  Channel4_ValueStatus := True,
                  Channel5_ValueStatus := True,
                  Channel6_ValueStatus := True,
                  Channel7_ValueStatus := True,
                  FIODia => "数据块_2"."F-DI_A21_1");
END_REGION

REGION Network 8: A21.2 诊断
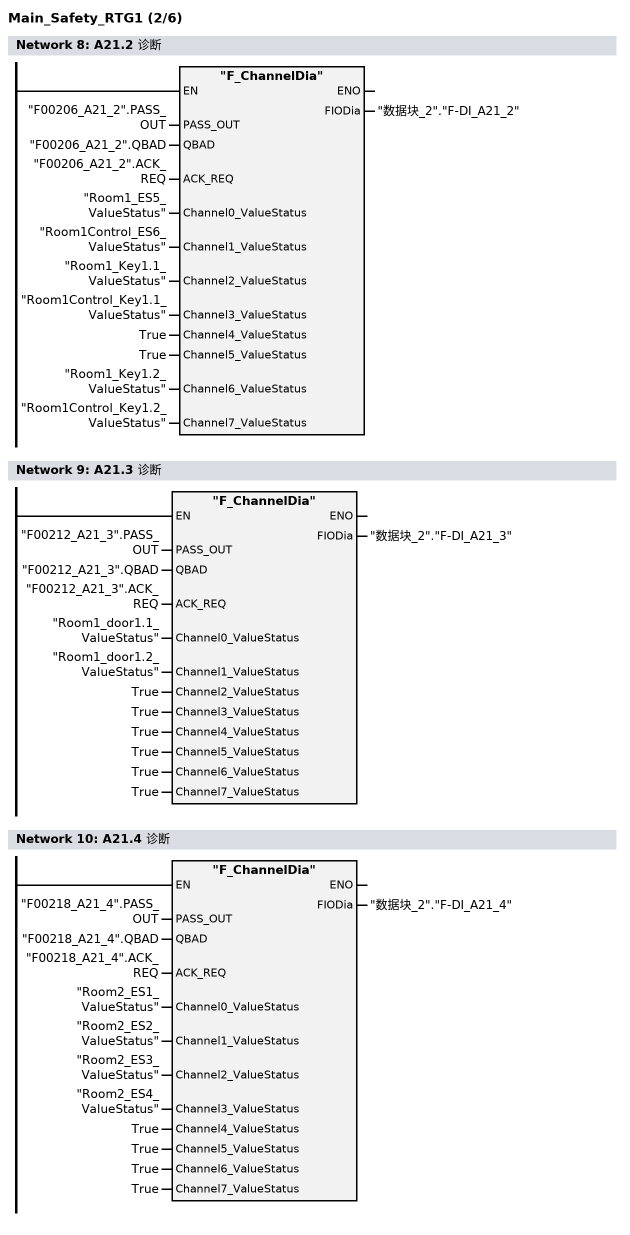
   RUNG wire#powerrail
      "F_ChannelDia"(PASS_OUT := "F00206_A21_2".PASS_OUT, QBAD := "F00206_A21_2".QBAD, ACK_REQ := "F00206_A21_2".ACK_REQ, Channel0_ValueStatus := "Room1_ES5_ValueStatus", Channel1_ValueStatus := "Room1Control_ES6_ValueStatus", Channel2_ValueStatus := "Room1_Key1.1_ValueStatus", Channel3_ValueStatus := "Room1Control_Key1.1_ValueStatus", Channel4_ValueStatus := True, Channel5_ValueStatus := True, Channel6_ValueStatus := "Room1_Key1.2_ValueStatus", Channel7_ValueStatus := "Room1Control_Key1.2_ValueStatus", FIODia => "数据块_2"."F-DI_A21_2")
   END_RUNG
   // the same network as SCL:
   "F_ChannelDia"(PASS_OUT := "F00206_A21_2".PASS_OUT,
                  QBAD := "F00206_A21_2".QBAD,
                  ACK_REQ := "F00206_A21_2".ACK_REQ,
                  Channel0_ValueStatus := "Room1_ES5_ValueStatus",
                  Channel1_ValueStatus := "Room1Control_ES6_ValueStatus",
                  Channel2_ValueStatus := "Room1_Key1.1_ValueStatus",
                  Channel3_ValueStatus := "Room1Control_Key1.1_ValueStatus",
                  Channel4_ValueStatus := True,
                  Channel5_ValueStatus := True,
                  Channel6_ValueStatus := "Room1_Key1.2_ValueStatus",
                  Channel7_ValueStatus := "Room1Control_Key1.2_ValueStatus",
                  FIODia => "数据块_2"."F-DI_A21_2");
END_REGION

REGION Network 9: A21.3 诊断
   RUNG wire#powerrail
      "F_ChannelDia"(PASS_OUT := "F00212_A21_3".PASS_OUT, QBAD := "F00212_A21_3".QBAD, ACK_REQ := "F00212_A21_3".ACK_REQ, Channel0_ValueStatus := "Room1_door1.1_ValueStatus", Channel1_ValueStatus := "Room1_door1.2_ValueStatus", Channel2_ValueStatus := True, Channel3_ValueStatus := True, Channel4_ValueStatus := True, Channel5_ValueStatus := True, Channel6_ValueStatus := True, Channel7_ValueStatus := True, FIODia => "数据块_2"."F-DI_A21_3")
   END_RUNG
   // the same network as SCL:
   "F_ChannelDia"(PASS_OUT := "F00212_A21_3".PASS_OUT,
                  QBAD := "F00212_A21_3".QBAD,
                  ACK_REQ := "F00212_A21_3".ACK_REQ,
                  Channel0_ValueStatus := "Room1_door1.1_ValueStatus",
                  Channel1_ValueStatus := "Room1_door1.2_ValueStatus",
                  Channel2_ValueStatus := True,
                  Channel3_ValueStatus := True,
                  Channel4_ValueStatus := True,
                  Channel5_ValueStatus := True,
                  Channel6_ValueStatus := True,
                  Channel7_ValueStatus := True,
                  FIODia => "数据块_2"."F-DI_A21_3");
END_REGION

REGION Network 10: A21.4 诊断
   RUNG wire#powerrail
      "F_ChannelDia"(PASS_OUT := "F00218_A21_4".PASS_OUT, QBAD := "F00218_A21_4".QBAD, ACK_REQ := "F00218_A21_4".ACK_REQ, Channel0_ValueStatus := "Room2_ES1_ValueStatus", Channel1_ValueStatus := "Room2_ES2_ValueStatus", Channel2_ValueStatus := "Room2_ES3_ValueStatus", Channel3_ValueStatus := "Room2_ES4_ValueStatus", Channel4_ValueStatus := True, Channel5_ValueStatus := True, Channel6_ValueStatus := True, Channel7_ValueStatus := True, FIODia => "数据块_2"."F-DI_A21_4")
   END_RUNG
   // the same network as SCL:
   "F_ChannelDia"(PASS_OUT := "F00218_A21_4".PASS_OUT,
                  QBAD := "F00218_A21_4".QBAD,
                  ACK_REQ := "F00218_A21_4".ACK_REQ,
                  Channel0_ValueStatus := "Room2_ES1_ValueStatus",
                  Channel1_ValueStatus := "Room2_ES2_ValueStatus",
                  Channel2_ValueStatus := "Room2_ES3_ValueStatus",
                  Channel3_ValueStatus := "Room2_ES4_ValueStatus",
                  Channel4_ValueStatus := True,
                  Channel5_ValueStatus := True,
                  Channel6_ValueStatus := True,
                  Channel7_ValueStatus := True,
                  FIODia => "数据块_2"."F-DI_A21_4");
END_REGION

REGION Network 11: A21.5 诊断
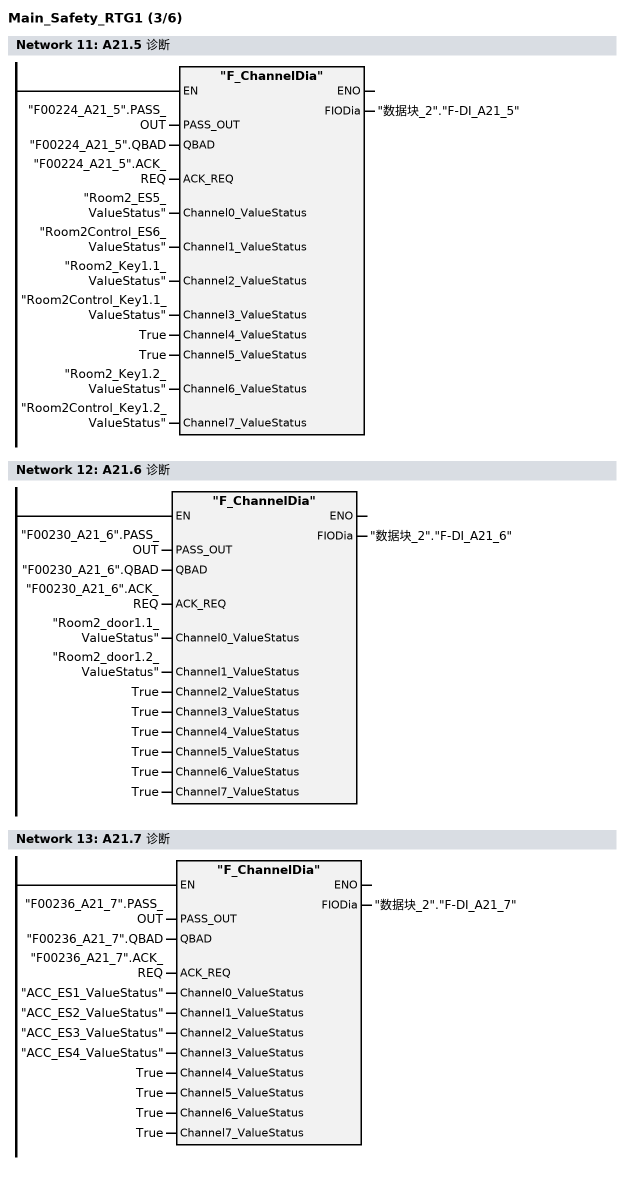
   RUNG wire#powerrail
      "F_ChannelDia"(PASS_OUT := "F00224_A21_5".PASS_OUT, QBAD := "F00224_A21_5".QBAD, ACK_REQ := "F00224_A21_5".ACK_REQ, Channel0_ValueStatus := "Room2_ES5_ValueStatus", Channel1_ValueStatus := "Room2Control_ES6_ValueStatus", Channel2_ValueStatus := "Room2_Key1.1_ValueStatus", Channel3_ValueStatus := "Room2Control_Key1.1_ValueStatus", Channel4_ValueStatus := True, Channel5_ValueStatus := True, Channel6_ValueStatus := "Room2_Key1.2_ValueStatus", Channel7_ValueStatus := "Room2Control_Key1.2_ValueStatus", FIODia => "数据块_2"."F-DI_A21_5")
   END_RUNG
   // the same network as SCL:
   "F_ChannelDia"(PASS_OUT := "F00224_A21_5".PASS_OUT,
                  QBAD := "F00224_A21_5".QBAD,
                  ACK_REQ := "F00224_A21_5".ACK_REQ,
                  Channel0_ValueStatus := "Room2_ES5_ValueStatus",
                  Channel1_ValueStatus := "Room2Control_ES6_ValueStatus",
                  Channel2_ValueStatus := "Room2_Key1.1_ValueStatus",
                  Channel3_ValueStatus := "Room2Control_Key1.1_ValueStatus",
                  Channel4_ValueStatus := True,
                  Channel5_ValueStatus := True,
                  Channel6_ValueStatus := "Room2_Key1.2_ValueStatus",
                  Channel7_ValueStatus := "Room2Control_Key1.2_ValueStatus",
                  FIODia => "数据块_2"."F-DI_A21_5");
END_REGION

REGION Network 12: A21.6 诊断
   RUNG wire#powerrail
      "F_ChannelDia"(PASS_OUT := "F00230_A21_6".PASS_OUT, QBAD := "F00230_A21_6".QBAD, ACK_REQ := "F00230_A21_6".ACK_REQ, Channel0_ValueStatus := "Room2_door1.1_ValueStatus", Channel1_ValueStatus := "Room2_door1.2_ValueStatus", Channel2_ValueStatus := True, Channel3_ValueStatus := True, Channel4_ValueStatus := True, Channel5_ValueStatus := True, Channel6_ValueStatus := True, Channel7_ValueStatus := True, FIODia => "数据块_2"."F-DI_A21_6")
   END_RUNG
   // the same network as SCL:
   "F_ChannelDia"(PASS_OUT := "F00230_A21_6".PASS_OUT,
                  QBAD := "F00230_A21_6".QBAD,
                  ACK_REQ := "F00230_A21_6".ACK_REQ,
                  Channel0_ValueStatus := "Room2_door1.1_ValueStatus",
                  Channel1_ValueStatus := "Room2_door1.2_ValueStatus",
                  Channel2_ValueStatus := True,
                  Channel3_ValueStatus := True,
                  Channel4_ValueStatus := True,
                  Channel5_ValueStatus := True,
                  Channel6_ValueStatus := True,
                  Channel7_ValueStatus := True,
                  FIODia => "数据块_2"."F-DI_A21_6");
END_REGION

REGION Network 13: A21.7 诊断
   RUNG wire#powerrail
      "F_ChannelDia"(PASS_OUT := "F00236_A21_7".PASS_OUT, QBAD := "F00236_A21_7".QBAD, ACK_REQ := "F00236_A21_7".ACK_REQ, Channel0_ValueStatus := "ACC_ES1_ValueStatus", Channel1_ValueStatus := "ACC_ES2_ValueStatus", Channel2_ValueStatus := "ACC_ES3_ValueStatus", Channel3_ValueStatus := "ACC_ES4_ValueStatus", Channel4_ValueStatus := True, Channel5_ValueStatus := True, Channel6_ValueStatus := True, Channel7_ValueStatus := True, FIODia => "数据块_2"."F-DI_A21_7")
   END_RUNG
   // the same network as SCL:
   "F_ChannelDia"(PASS_OUT := "F00236_A21_7".PASS_OUT,
                  QBAD := "F00236_A21_7".QBAD,
                  ACK_REQ := "F00236_A21_7".ACK_REQ,
                  Channel0_ValueStatus := "ACC_ES1_ValueStatus",
                  Channel1_ValueStatus := "ACC_ES2_ValueStatus",
                  Channel2_ValueStatus := "ACC_ES3_ValueStatus",
                  Channel3_ValueStatus := "ACC_ES4_ValueStatus",
                  Channel4_ValueStatus := True,
                  Channel5_ValueStatus := True,
                  Channel6_ValueStatus := True,
                  Channel7_ValueStatus := True,
                  FIODia => "数据块_2"."F-DI_A21_7");
END_REGION

REGION Network 14: A21.8 诊断
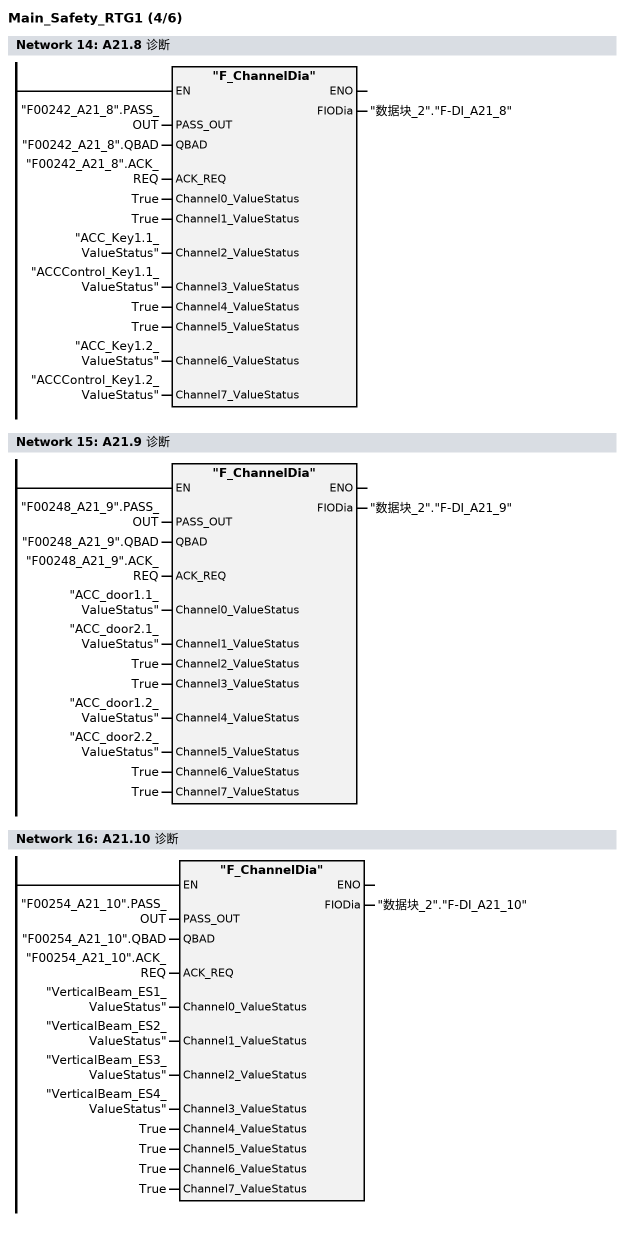
   RUNG wire#powerrail
      "F_ChannelDia"(PASS_OUT := "F00242_A21_8".PASS_OUT, QBAD := "F00242_A21_8".QBAD, ACK_REQ := "F00242_A21_8".ACK_REQ, Channel0_ValueStatus := True, Channel1_ValueStatus := True, Channel2_ValueStatus := "ACC_Key1.1_ValueStatus", Channel3_ValueStatus := "ACCControl_Key1.1_ValueStatus", Channel4_ValueStatus := True, Channel5_ValueStatus := True, Channel6_ValueStatus := "ACC_Key1.2_ValueStatus", Channel7_ValueStatus := "ACCControl_Key1.2_ValueStatus", FIODia => "数据块_2"."F-DI_A21_8")
   END_RUNG
   // the same network as SCL:
   "F_ChannelDia"(PASS_OUT := "F00242_A21_8".PASS_OUT,
                  QBAD := "F00242_A21_8".QBAD,
                  ACK_REQ := "F00242_A21_8".ACK_REQ,
                  Channel0_ValueStatus := True,
                  Channel1_ValueStatus := True,
                  Channel2_ValueStatus := "ACC_Key1.1_ValueStatus",
                  Channel3_ValueStatus := "ACCControl_Key1.1_ValueStatus",
                  Channel4_ValueStatus := True,
                  Channel5_ValueStatus := True,
                  Channel6_ValueStatus := "ACC_Key1.2_ValueStatus",
                  Channel7_ValueStatus := "ACCControl_Key1.2_ValueStatus",
                  FIODia => "数据块_2"."F-DI_A21_8");
END_REGION

REGION Network 15: A21.9 诊断
   RUNG wire#powerrail
      "F_ChannelDia"(PASS_OUT := "F00248_A21_9".PASS_OUT, QBAD := "F00248_A21_9".QBAD, ACK_REQ := "F00248_A21_9".ACK_REQ, Channel0_ValueStatus := "ACC_door1.1_ValueStatus", Channel1_ValueStatus := "ACC_door2.1_ValueStatus", Channel2_ValueStatus := True, Channel3_ValueStatus := True, Channel4_ValueStatus := "ACC_door1.2_ValueStatus", Channel5_ValueStatus := "ACC_door2.2_ValueStatus", Channel6_ValueStatus := True, Channel7_ValueStatus := True, FIODia => "数据块_2"."F-DI_A21_9")
   END_RUNG
   // the same network as SCL:
   "F_ChannelDia"(PASS_OUT := "F00248_A21_9".PASS_OUT,
                  QBAD := "F00248_A21_9".QBAD,
                  ACK_REQ := "F00248_A21_9".ACK_REQ,
                  Channel0_ValueStatus := "ACC_door1.1_ValueStatus",
                  Channel1_ValueStatus := "ACC_door2.1_ValueStatus",
                  Channel2_ValueStatus := True,
                  Channel3_ValueStatus := True,
                  Channel4_ValueStatus := "ACC_door1.2_ValueStatus",
                  Channel5_ValueStatus := "ACC_door2.2_ValueStatus",
                  Channel6_ValueStatus := True,
                  Channel7_ValueStatus := True,
                  FIODia => "数据块_2"."F-DI_A21_9");
END_REGION

REGION Network 16: A21.10 诊断
   RUNG wire#powerrail
      "F_ChannelDia"(PASS_OUT := "F00254_A21_10".PASS_OUT, QBAD := "F00254_A21_10".QBAD, ACK_REQ := "F00254_A21_10".ACK_REQ, Channel0_ValueStatus := "VerticalBeam_ES1_ValueStatus", Channel1_ValueStatus := "VerticalBeam_ES2_ValueStatus", Channel2_ValueStatus := "VerticalBeam_ES3_ValueStatus", Channel3_ValueStatus := "VerticalBeam_ES4_ValueStatus", Channel4_ValueStatus := True, Channel5_ValueStatus := True, Channel6_ValueStatus := True, Channel7_ValueStatus := True, FIODia => "数据块_2"."F-DI_A21_10")
   END_RUNG
   // the same network as SCL:
   "F_ChannelDia"(PASS_OUT := "F00254_A21_10".PASS_OUT,
                  QBAD := "F00254_A21_10".QBAD,
                  ACK_REQ := "F00254_A21_10".ACK_REQ,
                  Channel0_ValueStatus := "VerticalBeam_ES1_ValueStatus",
                  Channel1_ValueStatus := "VerticalBeam_ES2_ValueStatus",
                  Channel2_ValueStatus := "VerticalBeam_ES3_ValueStatus",
                  Channel3_ValueStatus := "VerticalBeam_ES4_ValueStatus",
                  Channel4_ValueStatus := True,
                  Channel5_ValueStatus := True,
                  Channel6_ValueStatus := True,
                  Channel7_ValueStatus := True,
                  FIODia => "数据块_2"."F-DI_A21_10");
END_REGION

REGION Network 17: A21.11 诊断
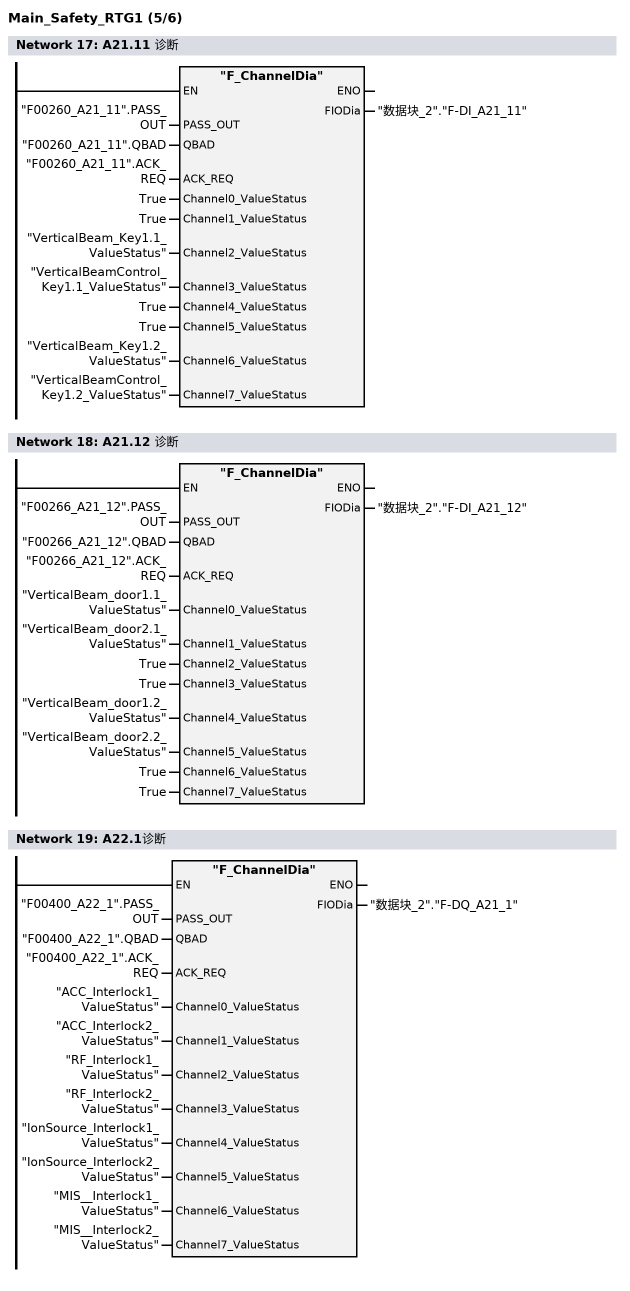
   RUNG wire#powerrail
      "F_ChannelDia"(PASS_OUT := "F00260_A21_11".PASS_OUT, QBAD := "F00260_A21_11".QBAD, ACK_REQ := "F00260_A21_11".ACK_REQ, Channel0_ValueStatus := True, Channel1_ValueStatus := True, Channel2_ValueStatus := "VerticalBeam_Key1.1_ValueStatus", Channel3_ValueStatus := "VerticalBeamControl_Key1.1_ValueStatus", Channel4_ValueStatus := True, Channel5_ValueStatus := True, Channel6_ValueStatus := "VerticalBeam_Key1.2_ValueStatus", Channel7_ValueStatus := "VerticalBeamControl_Key1.2_ValueStatus", FIODia => "数据块_2"."F-DI_A21_11")
   END_RUNG
   // the same network as SCL:
   "F_ChannelDia"(PASS_OUT := "F00260_A21_11".PASS_OUT,
                  QBAD := "F00260_A21_11".QBAD,
                  ACK_REQ := "F00260_A21_11".ACK_REQ,
                  Channel0_ValueStatus := True,
                  Channel1_ValueStatus := True,
                  Channel2_ValueStatus := "VerticalBeam_Key1.1_ValueStatus",
                  Channel3_ValueStatus := "VerticalBeamControl_Key1.1_ValueStatus",
                  Channel4_ValueStatus := True,
                  Channel5_ValueStatus := True,
                  Channel6_ValueStatus := "VerticalBeam_Key1.2_ValueStatus",
                  Channel7_ValueStatus := "VerticalBeamControl_Key1.2_ValueStatus",
                  FIODia => "数据块_2"."F-DI_A21_11");
END_REGION

REGION Network 18: A21.12 诊断
   RUNG wire#powerrail
      "F_ChannelDia"(PASS_OUT := "F00266_A21_12".PASS_OUT, QBAD := "F00266_A21_12".QBAD, ACK_REQ := "F00266_A21_12".ACK_REQ, Channel0_ValueStatus := "VerticalBeam_door1.1_ValueStatus", Channel1_ValueStatus := "VerticalBeam_door2.1_ValueStatus", Channel2_ValueStatus := True, Channel3_ValueStatus := True, Channel4_ValueStatus := "VerticalBeam_door1.2_ValueStatus", Channel5_ValueStatus := "VerticalBeam_door2.2_ValueStatus", Channel6_ValueStatus := True, Channel7_ValueStatus := True, FIODia => "数据块_2"."F-DI_A21_12")
   END_RUNG
   // the same network as SCL:
   "F_ChannelDia"(PASS_OUT := "F00266_A21_12".PASS_OUT,
                  QBAD := "F00266_A21_12".QBAD,
                  ACK_REQ := "F00266_A21_12".ACK_REQ,
                  Channel0_ValueStatus := "VerticalBeam_door1.1_ValueStatus",
                  Channel1_ValueStatus := "VerticalBeam_door2.1_ValueStatus",
                  Channel2_ValueStatus := True,
                  Channel3_ValueStatus := True,
                  Channel4_ValueStatus := "VerticalBeam_door1.2_ValueStatus",
                  Channel5_ValueStatus := "VerticalBeam_door2.2_ValueStatus",
                  Channel6_ValueStatus := True,
                  Channel7_ValueStatus := True,
                  FIODia => "数据块_2"."F-DI_A21_12");
END_REGION

REGION Network 19: A22.1诊断
   RUNG wire#powerrail
      "F_ChannelDia"(PASS_OUT := "F00400_A22_1".PASS_OUT, QBAD := "F00400_A22_1".QBAD, ACK_REQ := "F00400_A22_1".ACK_REQ, Channel0_ValueStatus := "ACC_Interlock1_ValueStatus", Channel1_ValueStatus := "ACC_Interlock2_ValueStatus", Channel2_ValueStatus := "RF_Interlock1_ValueStatus", Channel3_ValueStatus := "RF_Interlock2_ValueStatus", Channel4_ValueStatus := "IonSource_Interlock1_ValueStatus", Channel5_ValueStatus := "IonSource_Interlock2_ValueStatus", Channel6_ValueStatus := "MIS__Interlock1_ValueStatus", Channel7_ValueStatus := "MIS__Interlock2_ValueStatus", FIODia => "数据块_2"."F-DQ_A21_1")
   END_RUNG
   // the same network as SCL:
   "F_ChannelDia"(PASS_OUT := "F00400_A22_1".PASS_OUT,
                  QBAD := "F00400_A22_1".QBAD,
                  ACK_REQ := "F00400_A22_1".ACK_REQ,
                  Channel0_ValueStatus := "ACC_Interlock1_ValueStatus",
                  Channel1_ValueStatus := "ACC_Interlock2_ValueStatus",
                  Channel2_ValueStatus := "RF_Interlock1_ValueStatus",
                  Channel3_ValueStatus := "RF_Interlock2_ValueStatus",
                  Channel4_ValueStatus := "IonSource_Interlock1_ValueStatus",
                  Channel5_ValueStatus := "IonSource_Interlock2_ValueStatus",
                  Channel6_ValueStatus := "MIS__Interlock1_ValueStatus",
                  Channel7_ValueStatus := "MIS__Interlock2_ValueStatus",
                  FIODia => "数据块_2"."F-DQ_A21_1");
END_REGION

REGION Network 20: A22.2诊断
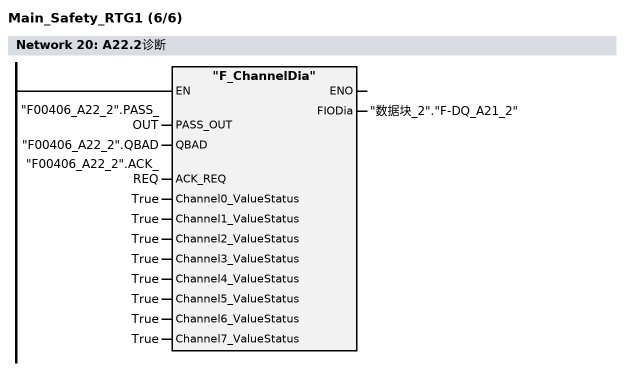
   RUNG wire#powerrail
      "F_ChannelDia"(PASS_OUT := "F00406_A22_2".PASS_OUT, QBAD := "F00406_A22_2".QBAD, ACK_REQ := "F00406_A22_2".ACK_REQ, Channel0_ValueStatus := True, Channel1_ValueStatus := True, Channel2_ValueStatus := True, Channel3_ValueStatus := True, Channel4_ValueStatus := True, Channel5_ValueStatus := True, Channel6_ValueStatus := True, Channel7_ValueStatus := True, FIODia => "数据块_2"."F-DQ_A21_2")
   END_RUNG
   // the same network as SCL:
   "F_ChannelDia"(PASS_OUT := "F00406_A22_2".PASS_OUT,
                  QBAD := "F00406_A22_2".QBAD,
                  ACK_REQ := "F00406_A22_2".ACK_REQ,
                  Channel0_ValueStatus := True,
                  Channel1_ValueStatus := True,
                  Channel2_ValueStatus := True,
                  Channel3_ValueStatus := True,
                  Channel4_ValueStatus := True,
                  Channel5_ValueStatus := True,
                  Channel6_ValueStatus := True,
                  Channel7_ValueStatus := True,
                  FIODia => "数据块_2"."F-DQ_A21_2");
END_REGION
END_FUNCTION_BLOCK

FUNCTION "Room1_Main" : Void   // FC4, LAD
{ S7_Optimized_Access := 'TRUE' }
VERSION : 0.1
// stored: AutoNumber true, IsIECCheckEnabled false, SetENOAutomatically false, UDAEnableTagReadback false
BEGIN

REGION Network 1: 区域搜索
